KUKA KRL program: MyProgram_340().src

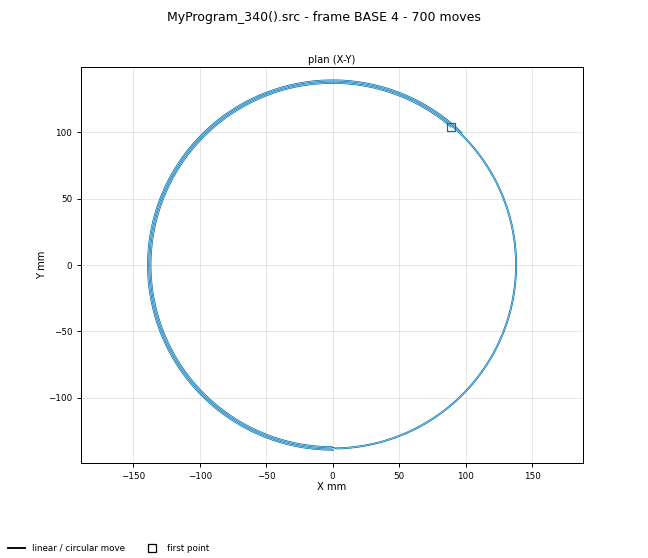
[picture p0: tool path of MyProgram_340().src in frame BASE 4, 700 of 700 moves have a stored position in this frame; points joined in program order, loops and branches not executed]
&ACCESS RVP
&REL 1
&PARAM TEMPLATE = C:\KRC\Roboter\Template\vorgabe
&PARAM EDITMASK = *
DEF MyProgram_340()
; ---- Setting reference (Base) ----
$BASE = BASE_DATA[4]

; --------------------------
; ---- Setting tool (TCP) ----
$TOOL = TOOL_DATA[3]
; --------------------------

$VEL.CP = VEL_APROX_PRINT
Startdeposition()
$VEL.CP = VEL_PRINT
LIN {X 89.0125,Y 103.7301,Z 191,A 47.9774,B 1.0012,C -0.0325,E1 1.1114,E2 406.47} C_DIS
LIN {X 85.5408,Y 106.6114,Z 191,A 49.6808,B 1.0011,C -0.0355,E1 1.1078,E2 404.7882} C_DIS
LIN {X 82.0051,Y 109.3546,Z 191,A 51.4263,B 1.001,C -0.0386,E1 1.1039,E2 403.0577} C_DIS
LIN {X 78.2991,Y 112.0376,Z 191,A 53.1641,B 1.0009,C -0.0415,E1 1.1,E2 401.3407} C_DIS
LIN {X 75.2781,Y 114.0891,Z 191,A 54.7295,B 1.0007,C -0.0444,E1 1.0963,E2 399.7713} C_DIS
LIN {X 72.4875,Y 115.8826,Z 191,A 55.8544,B 1.0007,C -0.0459,E1 1.0937,E2 398.6768} C_DIS
LIN {X 65.446,Y 119.9997,Z 191,A 58.9609,B 1.0005,C -0.0504,E1 1.0862,E2 395.6062} C_DIS
LIN {X 61.9887,Y 121.8193,Z 191,A 60.3832,B 1.0004,C -0.0523,E1 1.0827,E2 394.2083} C_DIS
LIN {X 59.3843,Y 123.111,Z 191,A 61.5861,B 1.0003,C -0.0541,E1 1.0796,E2 393.0073} C_DIS
LIN {X 56.2907,Y 124.556,Z 191,A 63.2488,B 1.0001,C -0.0571,E1 1.0753,E2 391.3188} C_DIS
LIN {X 52.6993,Y 126.1164,Z 191,A 64.3426,B 1.0001,C -0.0575,E1 1.0726,E2 390.2866} C_DIS
LIN {X 45.3684,Y 128.9368,Z 191,A 67.5319,B 0.9998,C -0.0616,E1 1.0643,E2 387.1097} C_DIS
LIN {X 41.7128,Y 130.1639,Z 191,A 68.9945,B 0.9998,C -0.0631,E1 1.0604,E2 385.6644} C_DIS
LIN {X 38.4614,Y 131.1614,Z 191,A 70.3424,B 0.9996,C -0.0645,E1 1.0567,E2 384.3254} C_DIS
LIN {X 34.8075,Y 132.1788,Z 191,A 71.8908,B 0.9996,C -0.0662,E1 1.0525,E2 382.7821} C_DIS
LIN {X 30.73,Y 133.1855,Z 191,A 73.5485,B 0.9994,C -0.0677,E1 1.048,E2 381.1362} C_DIS
LIN {X 27.316,Y 133.9271,Z 191,A 74.9001,B 0.9994,C -0.0688,E1 1.0443,E2 379.7974} C_DIS
LIN {X 24.0044,Y 134.5601,Z 191,A 76.1307,B 0.9994,C -0.0696,E1 1.041,E2 378.5872} C_DIS
LIN {X 21.0632,Y 135.0519,Z 191,A 77.6214,B 0.9992,C -0.0713,E1 1.0367,E2 377.0704} C_DIS
LIN {X 16.2963,Y 135.7096,Z 191,A 79.36,B 0.9992,C -0.0721,E1 1.0319,E2 375.3631} C_DIS
LIN {X 10.7417,Y 136.2638,Z 191,A 81.601,B 0.999,C -0.0735,E1 1.0257,E2 373.1338} C_DIS
LIN {X 3.1544,Y 136.6498,Z 191,A 84.6519,B 0.999,C -0.0749,E1 1.0171,E2 370.0986} C_DIS
LIN {X -4.6378,Y 136.6077,Z 191,A 88.9987,B 0.9986,C -0.0787,E1 1.0045,E2 365.6345} C_DIS
LIN {X -12.0307,Y 136.1551,Z 191,A 90.9637,B 0.9988,C -0.0769,E1 0.9993,E2 363.7961} C_DIS
LIN {X -15.8148,Y 135.7671,Z 191,A 92.6887,B 0.9988,C -0.0774,E1 0.9944,E2 362.0576} C_DIS
LIN {X -23.2946,Y 134.6872,Z 191,A 95.8708,B 0.9988,C -0.0774,E1 0.9855,E2 358.8755} C_DIS
LIN {X -27.1934,Y 133.9521,Z 191,A 97.4358,B 0.9988,C -0.0771,E1 0.9812,E2 357.3218} C_DIS
LIN {X -30.4676,Y 133.2454,Z 191,A 98.8461,B 0.9988,C -0.0769,E1 0.9773,E2 355.9115} C_DIS
LIN {X -34.0913,Y 132.3655,Z 191,A 100.4982,B 0.9988,C -0.0766,E1 0.9727,E2 354.2506} C_DIS
LIN {X -38.1454,Y 131.254,Z 191,A 102.2716,B 0.9988,C -0.0761,E1 0.9679,E2 352.4768} C_DIS
LIN {X -41.8854,Y 130.1088,Z 191,A 103.6911,B 0.9989,C -0.0751,E1 0.9642,E2 351.0819} C_DIS
LIN {X -46.7376,Y 128.4459,Z 191,A 106.4411,B 0.9989,C -0.0748,E1 0.9567,E2 348.2678} C_DIS
LIN {X -50.0052,Y 127.2098,Z 191,A 107.7565,B 0.999,C -0.0737,E1 0.9532,E2 346.9696} C_DIS
LIN {X -54.4673,Y 125.3632,Z 191,A 110.0747,B 0.999,C -0.0726,E1 0.9471,E2 344.6202} C_DIS
LIN {X -57.7457,Y 123.8877,Z 191,A 111.3528,B 0.9992,C -0.0712,E1 0.9439,E2 343.368} C_DIS
LIN {X -61.7186,Y 121.9568,Z 191,A 113.2508,B 0.9993,C -0.0696,E1 0.9391,E2 341.4659} C_DIS
LIN {X -65.1433,Y 120.1648,Z 191,A 115.3058,B 0.9993,C -0.0685,E1 0.9339,E2 339.3641} C_DIS
LIN {X -68.2953,Y 118.4015,Z 191,A 116.6428,B 0.9995,C -0.0668,E1 0.9306,E2 338.0475} C_DIS
LIN {X -71.0356,Y 116.7783,Z 191,A 118.4141,B 0.9995,C -0.0656,E1 0.9263,E2 336.2288} C_DIS
LIN {X -74.4665,Y 114.6204,Z 191,A 119.7536,B 0.9997,C -0.0634,E1 0.9232,E2 334.93} C_DIS
LIN {X -77.8426,Y 112.3553,Z 191,A 121.5206,B 0.9998,C -0.0613,E1 0.919,E2 333.1571} C_DIS
LIN {X -80.4484,Y 110.5045,Z 191,A 123.3051,B 0.9999,C -0.0597,E1 0.9149,E2 331.3241} C_DIS
LIN {X -86.3086,Y 105.9905,Z 191,A 126.4807,B 1.0002,C -0.0553,E1 0.9078,E2 328.1421} C_DIS
LIN {X -88.7872,Y 103.9233,Z 191,A 128.3952,B 1.0002,C -0.0534,E1 0.9036,E2 326.1654} C_DIS
LIN {X -92.1512,Y 100.9523,Z 191,A 129.7061,B 1.0005,C -0.0503,E1 0.901,E2 324.9197} C_DIS
LIN {X -97.6119,Y 95.6818,Z 191,A 133.23,B 1.0007,C -0.0449,E1 0.8938,E2 321.3597} C_DIS
LIN {X -100.937,Y 92.1667,Z 191,A 135.8857,B 1.0009,C -0.0412,E1 0.8886,E2 318.6342} C_DIS
LIN {X -106.4904,Y 85.6908,Z 191,A 139.6872,B 1.0011,C -0.0342,E1 0.8816,E2 314.8093} C_DIS
LIN {X -108.7863,Y 82.7573,Z 191,A 141.3018,B 1.0012,C -0.0311,E1 0.8789,E2 313.1896} C_DIS
LIN {X -111.015,Y 79.7425,Z 191,A 143.212,B 1.0013,C -0.0277,E1 0.8756,E2 311.2413} C_DIS
LIN {X -113.3974,Y 76.3169,Z 191,A 145.1171,B 1.0014,C -0.0239,E1 0.8726,E2 309.3194} C_DIS
LIN {X -115.7378,Y 72.7183,Z 191,A 147.066,B 1.0015,C -0.0198,E1 0.8696,E2 307.3543} C_DIS
LIN {X -118.0316,Y 68.9321,Z 191,A 149.3442,B 1.0016,C -0.0154,E1 0.8663,E2 305.0279} C_DIS
LIN {X -119.6578,Y 66.0693,Z 191,A 151.1723,B 1.0016,C -0.0119,E1 0.8637,E2 303.1479} C_DIS
LIN {X -121.3639,Y 62.8801,Z 191,A 152.6426,B 1.0016,C -0.0084,E1 0.8618,E2 301.684} C_DIS
LIN {X -122.9907,Y 59.6361,Z 191,A 154.354,B 1.0017,C -0.0046,E1 0.8597,E2 299.951} C_DIS
LIN {X -124.7758,Y 55.7992,Z 191,A 156.2284,B 1.0017,C -0.0001,E1 0.8575,E2 298.0657} C_DIS
LIN {X -126.2515,Y 52.3759,Z 191,A 158.1097,B 1.0017,C 0.004,E1 0.8554,E2 296.1474} C_DIS
LIN {X -127.8965,Y 48.2198,Z 191,A 160.229,B 1.0017,C 0.0089,E1 0.8532,E2 293.9998} C_DIS
LIN {X -129.0749,Y 44.9701,Z 191,A 161.9157,B 1.0017,C 0.0129,E1 0.8516,E2 292.2853} C_DIS
LIN {X -130.2137,Y 41.5569,Z 191,A 163.6416,B 1.0016,C 0.017,E1 0.8501,E2 290.534} C_DIS
LIN {X -131.1238,Y 38.5898,Z 191,A 165.1276,B 1.0016,C 0.0206,E1 0.8489,E2 289.0263} C_DIS
LIN {X -131.9252,Y 35.7585,Z 191,A 166.5518,B 1.0014,C 0.024,E1 0.8478,E2 287.5796} C_DIS
LIN {X -132.8248,Y 32.2526,Z 191,A 168.7786,B 1.0014,C 0.0287,E1 0.8463,E2 285.2663} C_DIS
LIN {X -133.6596,Y 28.5972,Z 191,A 170.156,B 1.0012,C 0.0328,E1 0.8455,E2 283.9139} C_DIS
LIN {X -134.4207,Y 24.7837,Z 191,A 172.2093,B 1.001,C 0.0376,E1 0.8444,E2 281.8092} C_DIS
LIN {X -135.0064,Y 21.3572,Z 191,A 173.7372,B 1.0009,C 0.0417,E1 0.8437,E2 280.2733} C_DIS
LIN {X -135.4771,Y 18.1315,Z 191,A 175.4147,B 1.0007,C 0.0458,E1 0.843,E2 278.5578} C_DIS
LIN {X -135.9257,Y 14.3847,Z 191,A 177.2703,B 1.0005,C 0.0504,E1 0.8424,E2 276.6687} C_DIS
LIN {X -136.3047,Y 10.1866,Z 191,A 179.2613,B 1.0002,C 0.0555,E1 0.842,E2 274.6504} C_DIS
LIN {X -136.5247,Y 6.6162,Z 191,A -178.9262,B 0.9999,C 0.06,E1 0.8417,E2 272.7991} C_DIS
LIN {X -136.6594,Y 2.6599,Z 191,A -177.0143,B 0.9996,C 0.0649,E1 0.8416,E2 270.856} C_DIS
LIN {X -136.6818,Y -1.0196,Z 191,A -175.0654,B 0.9993,C 0.0695,E1 0.8416,E2 268.8557} C_DIS
LIN {X -136.5818,Y -5.3018,Z 191,A -173.1233,B 0.9989,C 0.0747,E1 0.8417,E2 266.8957} C_DIS
LIN {X -136.3676,Y -9.3245,Z 191,A -171.0934,B 0.9985,C 0.0797,E1 0.8421,E2 264.8227} C_DIS
LIN {X -136.054,Y -13.1141,Z 191,A -169.2581,B 0.9982,C 0.0843,E1 0.8426,E2 262.9567} C_DIS
LIN {X -135.5716,Y -17.4107,Z 191,A -167.1462,B 0.9977,C 0.0896,E1 0.8433,E2 260.8066} C_DIS
LIN {X -135.0756,Y -20.9104,Z 191,A -165.3797,B 0.9973,C 0.0939,E1 0.844,E2 259.0034} C_DIS
LIN {X -134.3255,Y -25.287,Z 191,A -163.2215,B 0.9968,C 0.0992,E1 0.8451,E2 256.807} C_DIS
LIN {X -133.6562,Y -28.6131,Z 191,A -161.7639,B 0.9964,C 0.103,E1 0.8459,E2 255.3453} C_DIS
LIN {X -132.915,Y -31.8785,Z 191,A -160.1593,B 0.996,C 0.107,E1 0.847,E2 253.7147} C_DIS
LIN {X -132.2033,Y -34.7156,Z 191,A -158.4885,B 0.9956,C 0.1105,E1 0.8482,E2 251.9852} C_DIS
LIN {X -131.2438,Y -38.18,Z 191,A -156.9119,B 0.9952,C 0.1145,E1 0.8494,E2 250.4} C_DIS
LIN {X -130.259,Y -41.4151,Z 191,A -155.3551,B 0.9947,C 0.1183,E1 0.8507,E2 248.825} C_DIS
LIN {X -129.3087,Y -44.2956,Z 191,A -153.8993,B 0.9943,C 0.1217,E1 0.852,E2 247.345} C_DIS
LIN {X -127.3684,Y -49.597,Z 191,A -151.0547,B 0.9935,C 0.128,E1 0.8548,E2 244.4368} C_DIS
LIN {X -126.0875,Y -52.7686,Z 191,A -149.3641,B 0.993,C 0.1317,E1 0.8567,E2 242.7118} C_DIS
LIN {X -124.7202,Y -55.9236,Z 191,A -147.7644,B 0.9925,C 0.1353,E1 0.8585,E2 241.0911} C_DIS
LIN {X -123.4648,Y -58.6438,Z 191,A -146.2796,B 0.9921,C 0.1384,E1 0.8603,E2 239.5754} C_DIS
LIN {X -121.9116,Y -61.8075,Z 191,A -144.679,B 0.9916,C 0.142,E1 0.8623,E2 237.9583} C_DIS
LIN {X -120.1841,Y -65.1061,Z 191,A -142.4979,B 0.9911,C 0.1458,E1 0.8653,E2 235.6923} C_DIS
LIN {X -118.5495,Y -68.0385,Z 191,A -141.1245,B 0.9906,C 0.1489,E1 0.8672,E2 234.3241} C_DIS
LIN {X -116.0458,Y -72.2251,Z 191,A -138.8268,B 0.9899,C 0.1535,E1 0.8706,E2 231.9918} C_DIS
LIN {X -113.6068,Y -76.0041,Z 191,A -136.7006,B 0.9892,C 0.1576,E1 0.874,E2 229.8325} C_DIS
LIN {X -111.2543,Y -79.4078,Z 191,A -134.7546,B 0.9887,C 0.1612,E1 0.8772,E2 227.8574} C_DIS
LIN {X -108.5406,Y -83.0786,Z 191,A -132.6287,B 0.988,C 0.1651,E1 0.8808,E2 225.7021} C_DIS
LIN {X -105.6615,Y -86.7112,Z 191,A -130.4933,B 0.9874,C 0.1688,E1 0.8846,E2 223.54} C_DIS
LIN {X -102.7803,Y -90.1077,Z 191,A -128.4742,B 0.9868,C 0.1723,E1 0.8883,E2 221.4997} C_DIS
LIN {X -99.9949,Y -93.1886,Z 191,A -126.4868,B 0.9863,C 0.1753,E1 0.8922,E2 219.4776} C_DIS
LIN {X -96.802,Y -96.5015,Z 191,A -124.4491,B 0.9857,C 0.1786,E1 0.8962,E2 217.4246} C_DIS
LIN {X -91.9919,Y -101.0971,Z 191,A -121.3065,B 0.9849,C 0.1829,E1 0.9028,E2 214.232} C_DIS
LIN {X -88.5887,Y -104.092,Z 191,A -119.2485,B 0.9844,C 0.1857,E1 0.9072,E2 212.1516} C_DIS
LIN {X -85.0432,Y -107.0083,Z 191,A -117.1981,B 0.9839,C 0.1883,E1 0.9117,E2 210.0831} C_DIS
LIN {X -81.4237,Y -109.7877,Z 191,A -115.1197,B 0.9834,C 0.1907,E1 0.9165,E2 207.981} C_DIS
LIN {X -78.6696,Y -111.7775,Z 191,A -112.9292,B 0.9832,C 0.1917,E1 0.9218,E2 205.6802} C_DIS
LIN {X -74.0073,Y -114.918,Z 191,A -110.2765,B 0.9828,C 0.194,E1 0.9282,E2 202.9843} C_DIS
LIN {X -68.59,Y -118.2308,Z 191,A -108.2796,B 0.982,C 0.1977,E1 0.9328,E2 201.0832} C_DIS
LIN {X -64.6067,Y -120.4537,Z 191,A -106.1921,B 0.9817,C 0.1992,E1 0.9381,E2 198.9701} C_DIS
LIN {X -60.9145,Y -122.361,Z 191,A -104.507,B 0.9814,C 0.2008,E1 0.9423,E2 197.2928} C_DIS
LIN {X -55.0681,Y -125.1029,Z 191,A -101.7411,B 0.981,C 0.2028,E1 0.9494,E2 194.5179} C_DIS
LIN {X -48.4203,Y -127.8214,Z 191,A -98.6538,B 0.9806,C 0.2045,E1 0.9576,E2 191.4188} C_DIS
LIN {X -45.2797,Y -128.9675,Z 191,A -97.2652,B 0.9805,C 0.2052,E1 0.9612,E2 190.0317} C_DIS
LIN {X -41.8249,Y -130.1281,Z 191,A -95.648,B 0.9804,C 0.2057,E1 0.9656,E2 188.401} C_DIS
LIN {X -38.4661,Y -131.1601,Z 191,A -94.1345,B 0.9803,C 0.2062,E1 0.9697,E2 186.8811} C_DIS
LIN {X -35.798,Y -131.9146,Z 191,A -92.8618,B 0.9803,C 0.2062,E1 0.9732,E2 185.5921} C_DIS
LIN {X -32.0236,Y -132.88,Z 191,A -91.2701,B 0.9802,C 0.2067,E1 0.9776,E2 184.0058} C_DIS
LIN {X -28.5972,Y -133.6596,Z 191,A -89.7763,B 0.9802,C 0.2069,E1 0.9817,E2 182.5084} C_DIS
LIN {X -25.9354,Y -134.2016,Z 191,A -88.4583,B 0.9802,C 0.2066,E1 0.9855,E2 181.1639} C_DIS
LIN {X -20.2685,Y -135.175,Z 191,A -86.2694,B 0.9801,C 0.2071,E1 0.9915,E2 179.0062} C_DIS
LIN {X -15.9902,Y -135.7462,Z 191,A -84.4316,B 0.9801,C 0.2069,E1 0.9967,E2 177.1633} C_DIS
LIN {X -13.182,Y -136.0475,Z 191,A -82.9996,B 0.9803,C 0.206,E1 1.0008,E2 175.6947} C_DIS
LIN {X -7.968,Y -136.4529,Z 191,A -80.9818,B 0.9803,C 0.2059,E1 1.0064,E2 173.7012} C_DIS
LIN {X -0.5095,Y -136.684,Z 191,A -78.0357,B 0.9805,C 0.2052,E1 1.0147,E2 170.78} C_DIS
LIN {X -0.5095,Y -136.684,Z 191,A -78.0358,B 0.9805,C 0.2052,E1 1.0147,E2 170.7801} C_DIS
Enddeposition()
LIN {X 0.9755,Y -137.5796,Z 191,A -77.8874,B 0.9714,C 0.2064,E1 1.0061,E2 170.7271} C_DIS
Startdeposition()
$VEL.CP = VEL_PRINT
LIN {X -2.3504,Y -137.5636,Z 191,A -79.4321,B 0.9712,C 0.2074,E1 1.0017,E2 172.2957} C_DIS
LIN {X -6.1614,Y -137.4476,Z 191,A -80.9814,B 0.9712,C 0.2079,E1 0.9973,E2 173.8404} C_DIS
LIN {X -10.1773,Y -137.2067,Z 191,A -82.5541,B 0.9711,C 0.208,E1 0.9929,E2 175.3989} C_DIS
LIN {X -14.2933,Y -136.8397,Z 191,A -84.3553,B 0.971,C 0.2086,E1 0.9878,E2 177.2126} C_DIS
LIN {X -20.3097,Y -136.0782,Z 191,A -86.6928,B 0.971,C 0.2083,E1 0.9813,E2 179.524} C_DIS
LIN {X -26.9326,Y -134.9225,Z 191,A -89.4105,B 0.971,C 0.208,E1 0.9738,E2 182.231} C_DIS
LIN {X -30.869,Y -134.0758,Z 191,A -91.1981,B 0.971,C 0.208,E1 0.9688,E2 184.0353} C_DIS
LIN {X -34.03,Y -133.3085,Z 191,A -92.6122,B 0.9711,C 0.2079,E1 0.9649,E2 185.4586} C_DIS
LIN {X -37.2832,Y -132.4355,Z 191,A -94.0679,B 0.9711,C 0.2076,E1 0.9609,E2 186.9225} C_DIS
LIN {X -40.6978,Y -131.4269,Z 191,A -95.5338,B 0.9713,C 0.207,E1 0.9569,E2 188.3864} C_DIS
LIN {X -43.6182,Y -130.486,Z 191,A -96.8165,B 0.9714,C 0.2064,E1 0.9535,E2 189.6703} C_DIS
LIN {X -46.7356,Y -129.4021,Z 191,A -98.3193,B 0.9715,C 0.206,E1 0.9494,E2 191.1921} C_DIS
LIN {X -50.5842,Y -127.9491,Z 191,A -100.2988,B 0.9716,C 0.2055,E1 0.9441,E2 193.2105} C_DIS
LIN {X -54.8307,Y -126.1854,Z 191,A -101.9447,B 0.972,C 0.2038,E1 0.9399,E2 194.818} C_DIS
LIN {X -57.6498,Y -124.9224,Z 191,A -103.437,B 0.9721,C 0.2031,E1 0.936,E2 196.3404} C_DIS
LIN {X -61.24,Y -123.2028,Z 191,A -105.0696,B 0.9724,C 0.2018,E1 0.9319,E2 197.9697} C_DIS
LIN {X -64.6588,Y -121.4452,Z 191,A -106.8458,B 0.9727,C 0.2006,E1 0.9274,E2 199.7715} C_DIS
LIN {X -68.4652,Y -119.3411,Z 191,A -108.7461,B 0.973,C 0.1989,E1 0.9226,E2 201.6849} C_DIS
LIN {X -73.0298,Y -116.6039,Z 191,A -111.0777,B 0.9734,C 0.1967,E1 0.917,E2 204.0335} C_DIS
LIN {X -76.7762,Y -114.172,Z 191,A -113.3045,B 0.9738,C 0.1949,E1 0.9116,E2 206.313} C_DIS
LIN {X -79.5332,Y -112.2684,Z 191,A -114.5548,B 0.9742,C 0.193,E1 0.9088,E2 207.5427} C_DIS
LIN {X -82.9847,Y -109.7415,Z 191,A -116.466,B 0.9746,C 0.1908,E1 0.9044,E2 209.4725} C_DIS
LIN {X -86.4102,Y -107.0651,Z 191,A -118.4124,B 0.9751,C 0.1883,E1 0.9001,E2 211.4383} C_DIS
LIN {X -89.5447,Y -104.4581,Z 191,A -120.3137,B 0.9755,C 0.186,E1 0.8959,E2 213.3686} C_DIS
LIN {X -93.0211,Y -101.3742,Z 191,A -122.5042,B 0.9761,C 0.1831,E1 0.8913,E2 215.5953} C_DIS
LIN {X -96.7246,Y -97.8475,Z 191,A -124.6857,B 0.9767,C 0.1796,E1 0.8868,E2 217.7841} C_DIS
LIN {X -99.6065,Y -94.9117,Z 191,A -126.588,B 0.9773,C 0.1767,E1 0.8831,E2 219.7129} C_DIS
LIN {X -102.6845,Y -91.573,Z 191,A -128.6464,B 0.9779,C 0.1734,E1 0.8791,E2 221.7946} C_DIS
LIN {X -105.6134,Y -88.1791,Z 191,A -130.7495,B 0.9785,C 0.1699,E1 0.8752,E2 223.9307} C_DIS
LIN {X -108.4646,Y -84.6479,Z 191,A -132.8938,B 0.9791,C 0.1662,E1 0.8714,E2 226.1104} C_DIS
LIN {X -111.2531,Y -80.9472,Z 191,A -135.0363,B 0.9798,C 0.1623,E1 0.8678,E2 228.2822} C_DIS
LIN {X -113.8906,Y -77.1919,Z 191,A -137.175,B 0.9804,C 0.1583,E1 0.8643,E2 230.4522} C_DIS
LIN {X -116.3526,Y -73.4284,Z 191,A -139.3153,B 0.9811,C 0.1542,E1 0.861,E2 232.629} C_DIS
LIN {X -119.0033,Y -69.0499,Z 191,A -142.5443,B 0.9818,C 0.1492,E1 0.8563,E2 236.0081} C_DIS
LIN {X -121.9972,Y -63.6076,Z 191,A -144.5104,B 0.9827,C 0.1433,E1 0.8538,E2 237.8887} C_DIS
LIN {X -123.5368,Y -60.5629,Z 191,A -146.1854,B 0.9832,C 0.1399,E1 0.8516,E2 239.598} C_DIS
LIN {X -125.253,Y -56.9339,Z 191,A -148.2535,B 0.9838,C 0.1356,E1 0.8491,E2 241.7196} C_DIS
LIN {X -127.0422,Y -52.8152,Z 191,A -150.2585,B 0.9844,C 0.131,E1 0.8469,E2 243.7423} C_DIS
LIN {X -128.8535,Y -48.2274,Z 191,A -152.6351,B 0.9851,C 0.1256,E1 0.8445,E2 246.1617} C_DIS
LIN {X -130.1279,Y -44.6768,Z 191,A -154.3839,B 0.9857,C 0.1215,E1 0.8428,E2 247.9338} C_DIS
LIN {X -131.161,Y -41.5458,Z 191,A -155.925,B 0.9861,C 0.1178,E1 0.8415,E2 249.4969} C_DIS
LIN {X -132.1072,Y -38.4304,Z 191,A -157.5422,B 0.9865,C 0.1141,E1 0.8402,E2 251.1486} C_DIS
LIN {X -133.1124,Y -34.795,Z 191,A -159.3155,B 0.987,C 0.1098,E1 0.8389,E2 252.9482} C_DIS
LIN {X -133.7924,Y -32.0747,Z 191,A -160.6918,B 0.9874,C 0.1065,E1 0.8379,E2 254.3516} C_DIS
LIN {X -134.4829,Y -29.0433,Z 191,A -162.235,B 0.9878,C 0.1028,E1 0.837,E2 255.9272} C_DIS
LIN {X -135.2705,Y -25.1312,Z 191,A -164.3349,B 0.9883,C 0.098,E1 0.8358,E2 258.084} C_DIS
LIN {X -135.9783,Y -20.9551,Z 191,A -166.1966,B 0.9887,C 0.0931,E1 0.835,E2 259.9576} C_DIS
LIN {X -136.4504,Y -17.6228,Z 191,A -167.9204,B 0.9891,C 0.0889,E1 0.8343,E2 261.7228} C_DIS
LIN {X -136.9391,Y -13.301,Z 191,A -170.0176,B 0.9896,C 0.0837,E1 0.8337,E2 263.8562} C_DIS
LIN {X -137.2547,Y -9.5192,Z 191,A -171.9652,B 0.99,C 0.079,E1 0.8333,E2 265.8505} C_DIS
LIN {X -137.4766,Y -5.4259,Z 191,A -173.8399,B 0.9904,C 0.074,E1 0.833,E2 267.7458} C_DIS
LIN {X -137.5778,Y -1.4513,Z 191,A -175.8623,B 0.9907,C 0.0691,E1 0.833,E2 269.8142} C_DIS
LIN {X -137.5571,Y 2.7372,Z 191,A -177.8981,B 0.9911,C 0.0639,E1 0.833,E2 271.8861} C_DIS
LIN {X -137.416,Y 6.7903,Z 191,A -179.8134,B 0.9914,C 0.059,E1 0.8332,E2 273.8291} C_DIS
LIN {X -137.1733,Y 10.6343,Z 191,A 178.1911,B 0.9916,C 0.0542,E1 0.8336,E2 275.873} C_DIS
LIN {X -136.7905,Y 14.7502,Z 191,A 176.3408,B 0.9919,C 0.0493,E1 0.8341,E2 277.7383} C_DIS
LIN {X -136.3259,Y 18.5724,Z 191,A 174.2864,B 0.9921,C 0.0444,E1 0.8349,E2 279.848} C_DIS
LIN {X -135.7059,Y 22.6516,Z 191,A 172.4219,B 0.9923,C 0.0395,E1 0.8357,E2 281.7295} C_DIS
LIN {X -135.0578,Y 26.244,Z 191,A 170.6382,B 0.9925,C 0.0351,E1 0.8367,E2 283.5448} C_DIS
LIN {X -134.107,Y 30.7327,Z 191,A 168.39,B 0.9927,C 0.0297,E1 0.838,E2 285.8333} C_DIS
LIN {X -133.0599,Y 34.9919,Z 191,A 166.3658,B 0.9928,C 0.0246,E1 0.8394,E2 287.8805} C_DIS
LIN {X -132.1069,Y 38.4315,Z 191,A 164.4992,B 0.9929,C 0.0203,E1 0.8409,E2 289.7922} C_DIS
LIN {X -130.9132,Y 42.3214,Z 191,A 162.6742,B 0.9929,C 0.0157,E1 0.8424,E2 291.632} C_DIS
LIN {X -129.86,Y 45.4498,Z 191,A 161.0565,B 0.993,C 0.012,E1 0.8439,E2 293.278} C_DIS
LIN {X -128.7512,Y 48.5005,Z 191,A 159.4542,B 0.993,C 0.0083,E1 0.8455,E2 294.9094} C_DIS
LIN {X -127.3455,Y 52.0838,Z 191,A 157.6483,B 0.9931,C 0.0041,E1 0.8474,E2 296.7386} C_DIS
LIN {X -125.8846,Y 55.5219,Z 191,A 155.6562,B 0.9931,C -0.0001,E1 0.8497,E2 298.7813} C_DIS
LIN {X -123.9004,Y 59.8173,Z 191,A 153.6151,B 0.9931,C -0.0049,E1 0.8521,E2 300.8295} C_DIS
LIN {X -122.4671,Y 62.6977,Z 191,A 152.0069,B 0.9931,C -0.0083,E1 0.8542,E2 302.4682} C_DIS
LIN {X -120.1746,Y 66.9917,Z 191,A 149.6109,B 0.9931,C -0.0133,E1 0.8575,E2 304.906} C_DIS
LIN {X -117.1207,Y 72.1975,Z 191,A 146.7692,B 0.9929,C -0.0191,E1 0.8616,E2 307.7841} C_DIS
LIN {X -114.6585,Y 76.0476,Z 191,A 144.6065,B 0.9929,C -0.0234,E1 0.865,E2 309.9754} C_DIS
LIN {X -112.1096,Y 79.7571,Z 191,A 142.5051,B 0.9927,C -0.0275,E1 0.8684,E2 312.1015} C_DIS
LIN {X -108.8533,Y 84.1466,Z 191,A 140.1427,B 0.9926,C -0.0322,E1 0.8724,E2 314.4724} C_DIS
LIN {X -105.323,Y 88.5252,Z 191,A 137.2526,B 0.9924,C -0.0369,E1 0.8776,E2 317.423} C_DIS
LIN {X -102.4692,Y 91.8135,Z 191,A 134.6875,B 0.9923,C -0.0404,E1 0.8826,E2 320.0708} C_DIS
LIN {X -98.7949,Y 95.7561,Z 191,A 133.367,B 0.9921,C -0.0444,E1 0.885,E2 321.2868} C_DIS
LIN {X -95.3607,Y 99.1774,Z 191,A 130.6309,B 0.992,C -0.0478,E1 0.8906,E2 324.102} C_DIS
LIN {X -91.3994,Y 102.839,Z 191,A 127.6625,B 0.9918,C -0.0513,E1 0.897,E2 327.1485} C_DIS
LIN {X -87.7377,Y 105.9799,Z 191,A 126.1159,B 0.9916,C -0.0544,E1 0.9002,E2 328.6432} C_DIS
LIN {X -82.2759,Y 110.274,Z 191,A 122.4127,B 0.9914,C -0.0582,E1 0.9087,E2 332.4332} C_DIS
LIN {X -78.5502,Y 112.958,Z 191,A 120.9733,B 0.9913,C -0.0608,E1 0.9119,E2 333.82} C_DIS
LIN {X -75.2948,Y 115.1544,Z 191,A 119.0116,B 0.9911,C -0.0626,E1 0.9166,E2 335.8164} C_DIS
LIN {X -71.5352,Y 117.5267,Z 191,A 117.0965,B 0.9911,C -0.0647,E1 0.9212,E2 337.7373} C_DIS
LIN {X -67.6499,Y 119.8049,Z 191,A 115.1076,B 0.9909,C -0.0665,E1 0.9261,E2 339.7375} C_DIS
LIN {X -63.7058,Y 121.9456,Z 191,A 113.2532,B 0.9908,C -0.0683,E1 0.9307,E2 341.5891} C_DIS
LIN {X -60.3355,Y 123.649,Z 191,A 111.5289,B 0.9907,C -0.0695,E1 0.9351,E2 343.3291} C_DIS
LIN {X -56.6215,Y 125.3928,Z 191,A 109.2716,B 0.9907,C -0.0702,E1 0.9411,E2 345.6442} C_DIS
LIN {X -52.2336,Y 127.2849,Z 191,A 107.7938,B 0.9905,C -0.0721,E1 0.9448,E2 347.0662} C_DIS
LIN {X -48.6101,Y 128.7102,Z 191,A 105.2683,B 0.9905,C -0.072,E1 0.9517,E2 349.6873} C_DIS
LIN {X -42.8275,Y 130.7493,Z 191,A 103.5296,B 0.9903,C -0.0743,E1 0.9561,E2 351.338} C_DIS
LIN {X -39.9991,Y 131.6407,Z 191,A 102.1985,B 0.9903,C -0.0746,E1 0.9597,E2 352.6787} C_DIS
LIN {X -36.7199,Y 132.593,Z 191,A 100.8049,B 0.9903,C -0.0752,E1 0.9635,E2 354.0685} C_DIS
LIN {X -33.2062,Y 133.5176,Z 191,A 99.2577,B 0.9903,C -0.0755,E1 0.9678,E2 355.6187} C_DIS
LIN {X -30.1359,Y 134.2433,Z 191,A 97.9714,B 0.9903,C -0.0758,E1 0.9713,E2 356.9015} C_DIS
LIN {X -27.1204,Y 134.8843,Z 191,A 96.6055,B 0.9903,C -0.0758,E1 0.9751,E2 358.2755} C_DIS
LIN {X -22.8887,Y 135.6664,Z 191,A 94.6325,B 0.9903,C -0.0756,E1 0.9807,E2 360.2671} C_DIS
LIN {X -16.2805,Y 136.6168,Z 191,A 92.0873,B 0.9903,C -0.0758,E1 0.9877,E2 362.7859} C_DIS
LIN {X -12.9872,Y 136.9693,Z 191,A 90.7086,B 0.9903,C -0.0756,E1 0.9916,E2 364.1639} C_DIS
LIN {X -9.1202,Y 137.2825,Z 191,A 88.5737,B 0.9903,C -0.0741,E1 0.9978,E2 366.3537} C_DIS
LIN {X -4.5471,Y 137.5104,Z 191,A 87.2726,B 0.9903,C -0.0748,E1 1.0013,E2 367.5893} C_DIS
LIN {X 2.4832,Y 137.5614,Z 191,A 84.4448,B 0.9903,C -0.0737,E1 1.0093,E2 370.4052} C_DIS
LIN {X 5.7855,Y 137.4626,Z 191,A 83.0466,B 0.9904,C -0.073,E1 1.0132,E2 371.8053} C_DIS
LIN {X 8.6467,Y 137.3117,Z 191,A 81.8644,B 0.9904,C -0.0723,E1 1.0165,E2 372.9859} C_DIS
LIN {X 12.6768,Y 136.9991,Z 191,A 80.0333,B 0.9906,C -0.0708,E1 1.0217,E2 374.8324} C_DIS
LIN {X 17.0816,Y 136.5213,Z 191,A 78.4841,B 0.9906,C -0.0702,E1 1.026,E2 376.3492} C_DIS
LIN {X 23.4637,Y 135.5701,Z 191,A 75.9145,B 0.9908,C -0.0682,E1 1.0331,E2 378.9053} C_DIS
LIN {X 27.2464,Y 134.8586,Z 191,A 74.3537,B 0.9908,C -0.0668,E1 1.0375,E2 380.461} C_DIS
LIN {X 30.6029,Y 134.1366,Z 191,A 72.9821,B 0.9909,C -0.0656,E1 1.0412,E2 381.8258} C_DIS
LIN {X 34.149,Y 133.2783,Z 191,A 71.5276,B 0.991,C -0.0641,E1 1.0452,E2 383.2728} C_DIS
LIN {X 37.5501,Y 132.3609,Z 191,A 70.2116,B 0.9911,C -0.0629,E1 1.0487,E2 384.572} C_DIS
LIN {X 40.3296,Y 131.5396,Z 191,A 69.0293,B 0.9912,C -0.0616,E1 1.0519,E2 385.7513} C_DIS
LIN {X 43.6605,Y 130.472,Z 191,A 67.6613,B 0.9912,C -0.0601,E1 1.0555,E2 387.1093} C_DIS
LIN {X 47.3979,Y 129.163,Z 191,A 65.88,B 0.9915,C -0.0574,E1 1.0603,E2 388.9049} C_DIS
LIN {X 51.5423,Y 127.5638,Z 191,A 64.4,B 0.9915,C -0.0561,E1 1.0641,E2 390.3436} C_DIS
LIN {X 55.1122,Y 126.0637,Z 191,A 62.8498,B 0.9916,C -0.054,E1 1.0681,E2 391.8868} C_DIS
LIN {X 58.025,Y 124.7489,Z 191,A 61.6509,B 0.9917,C -0.0525,E1 1.0711,E2 393.0708} C_DIS
LIN {X 61.331,Y 123.1579,Z 191,A 60.2491,B 0.9918,C -0.0506,E1 1.0746,E2 394.4583} C_DIS
LIN {X 65.1031,Y 121.2074,Z 191,A 58.5274,B 0.992,C -0.0479,E1 1.0789,E2 396.1747} C_DIS
LIN {X 69.6354,Y 118.6616,Z 191,A 56.7498,B 0.992,C -0.0457,E1 1.0832,E2 397.9087} C_DIS
LIN {X 72.4509,Y 116.9641,Z 191,A 55.2563,B 0.9922,C -0.0428,E1 1.0868,E2 399.4161} C_DIS
LIN {X 76.2951,Y 114.4933,Z 191,A 53.5365,B 0.9923,C -0.0401,E1 1.0908,E2 401.1151} C_DIS
LIN {X 80.1583,Y 111.8227,Z 191,A 51.7644,B 0.9924,C -0.0371,E1 1.0948,E2 402.8663} C_DIS
LIN {X 83.872,Y 109.0655,Z 191,A 50.0063,B 0.9925,C -0.0341,E1 1.0987,E2 404.6054} C_DIS
LIN {X 87.2973,Y 106.3434,Z 191,A 48.3731,B 0.9926,C -0.0312,E1 1.1022,E2 406.2171} C_DIS
LIN {X 90.7316,Y 103.429,Z 191,A 46.6587,B 0.9927,C -0.0281,E1 1.1058,E2 407.9131} C_DIS
LIN {X 93.954,Y 100.5105,Z 191,A 45.0724,B 0.9927,C -0.0252,E1 1.1091,E2 409.4737} C_DIS
LIN {X 97.0603,Y 97.5139,Z 191,A 43.4133,B 0.9929,C -0.022,E1 1.1124,E2 411.1169} C_DIS
LIN {X 100.2727,Y 94.2078,Z 191,A 41.6823,B 0.9929,C -0.0186,E1 1.1157,E2 412.8262} C_DIS
LIN {X 103.2679,Y 90.9146,Z 191,A 40.02,B 0.9929,C -0.0152,E1 1.1188,E2 414.4664} C_DIS
LIN {X 106.2288,Y 87.4372,Z 191,A 38.3589,B 0.993,C -0.0119,E1 1.1217,E2 416.0996} C_DIS
LIN {X 108.9095,Y 84.074,Z 191,A 36.7417,B 0.993,C -0.0085,E1 1.1245,E2 417.6966} C_DIS
LIN {X 111.5028,Y 80.6027,Z 191,A 35.1119,B 0.9931,C -0.0051,E1 1.1271,E2 419.3062} C_DIS
LIN {X 114.1371,Y 76.8277,Z 191,A 33.349,B 0.9931,C -0.0011,E1 1.1299,E2 421.0512} C_DIS
LIN {X 116.5474,Y 73.1198,Z 191,A 31.7983,B 0.9931,C 0.002,E1 1.1322,E2 422.5676} C_DIS
LIN {X 118.8132,Y 69.3773,Z 191,A 30.1058,B 0.9931,C 0.006,E1 1.1346,E2 424.2451} C_DIS
LIN {X 121.0286,Y 65.436,Z 191,A 28.4668,B 0.9931,C 0.0096,E1 1.1368,E2 425.8554} C_DIS
LIN {X 122.9821,Y 61.6861,Z 191,A 26.9917,B 0.9931,C 0.0127,E1 1.1386,E2 427.2964} C_DIS
LIN {X 124.757,Y 58.0074,Z 191,A 25.3815,B 0.993,C 0.0166,E1 1.1405,E2 428.8961} C_DIS
LIN {X 126.6075,Y 53.8546,Z 191,A 23.8342,B 0.993,C 0.0199,E1 1.1422,E2 430.402} C_DIS
LIN {X 128.1012,Y 50.1931,Z 191,A 22.1781,B 0.9928,C 0.0243,E1 1.1439,E2 432.0597} C_DIS
LIN {X 130.0598,Y 44.8735,Z 191,A 20.2967,B 0.9928,C 0.0281,E1 1.1456,E2 433.8832} C_DIS
LIN {X 131.178,Y 41.4923,Z 191,A 18.9949,B 0.9926,C 0.0312,E1 1.1467,E2 435.1631} C_DIS
LIN {X 132.0841,Y 38.5092,Z 191,A 17.8663,B 0.9926,C 0.0339,E1 1.1476,E2 436.2712} C_DIS
LIN {X 132.9957,Y 35.2328,Z 191,A 16.6235,B 0.9924,C 0.0368,E1 1.1485,E2 437.493} C_DIS
LIN {X 133.8062,Y 32.0173,Z 191,A 15.3967,B 0.9924,C 0.0398,E1 1.1493,E2 438.7012} C_DIS
LIN {X 134.6323,Y 28.3513,Z 191,A 14.0446,B 0.9922,C 0.043,E1 1.1501,E2 440.0274} C_DIS
LIN {X 135.3181,Y 24.8718,Z 191,A 12.2949,B 0.9919,C 0.0485,E1 1.151,E2 441.8118} C_DIS
LIN {X 136.0408,Y 20.5514,Z 191,A 11.2082,B 0.9919,C 0.0497,E1 1.1515,E2 442.8067} C_DIS
LIN {X 136.5706,Y 16.6678,Z 191,A 9.3411,B 0.9916,C 0.0554,E1 1.1521,E2 444.7043} C_DIS
LIN {X 136.9914,Y 12.7568,Z 191,A 8.2247,B 0.9915,C 0.0572,E1 1.1524,E2 445.7554} C_DIS
LIN {X 137.4528,Y 6.0368,Z 191,A 5.8564,B 0.9911,C 0.0628,E1 1.1528,E2 448.0694} C_DIS
LIN {X 137.5564,Y 2.7845,Z 191,A 4.2134,B 0.9908,C 0.0681,E1 1.1529,E2 449.75} C_DIS
LIN {X 137.5775,Y -1.4988,Z 191,A 3.0781,B 0.9907,C 0.0696,E1 1.1529,E2 450.8031} C_DIS
LIN {X 137.4312,Y -6.4873,Z 191,A 1.3571,B 0.9904,C 0.0735,E1 1.1528,E2 452.479} C_DIS
LIN {X 137.218,Y -10.0226,Z 191,A -0.092,B 0.9901,C 0.0774,E1 1.1525,E2 453.9256} C_DIS
LIN {X 136.9084,Y -13.6213,Z 191,A -1.339,B 0.9899,C 0.0803,E1 1.1522,E2 455.1401} C_DIS
LIN {X 136.5553,Y -16.7959,Z 191,A -2.9154,B 0.9894,C 0.0853,E1 1.1516,E2 456.7494} C_DIS
LIN {X 136.0169,Y -20.7054,Z 191,A -3.8611,B 0.9894,C 0.0861,E1 1.1513,E2 457.6048} C_DIS
LIN {X 135.4711,Y -24.0172,Z 191,A -5.2542,B 0.989,C 0.0899,E1 1.1507,E2 458.9982} C_DIS
LIN {X 134.7817,Y -27.6244,Z 191,A -6.6092,B 0.9887,C 0.0932,E1 1.1499,E2 460.3312} C_DIS
LIN {X 134.0208,Y -31.11,Z 191,A -7.8746,B 0.9885,C 0.0961,E1 1.1492,E2 461.5684} C_DIS
LIN {X 133.0231,Y -35.13,Z 191,A -9.4164,B 0.9881,C 0.0998,E1 1.1481,E2 463.0871} C_DIS
LIN {X 132.0785,Y -38.5283,Z 191,A -10.7105,B 0.9878,C 0.1029,E1 1.1471,E2 464.3588} C_DIS
LIN {X 130.8702,Y -42.4555,Z 191,A -12.4475,B 0.9873,C 0.1076,E1 1.1457,E2 466.1005} C_DIS
LIN {X 129.8042,Y -45.6107,Z 191,A -13.3938,B 0.9871,C 0.109,E1 1.1449,E2 466.9889} C_DIS
LIN {X 128.6922,Y -48.6581,Z 191,A -14.6459,B 0.9868,C 0.112,E1 1.1436,E2 468.2286} C_DIS
LIN {X 127.4906,Y -51.7238,Z 191,A -15.7881,B 0.9865,C 0.1145,E1 1.1425,E2 469.3409} C_DIS
LIN {X 125.9612,Y -55.3494,Z 191,A -17.2542,B 0.9861,C 0.1178,E1 1.1409,E2 470.785} C_DIS
LIN {X 124.7852,Y -57.9466,Z 191,A -18.3351,B 0.9858,C 0.1204,E1 1.1397,E2 471.8522} C_DIS
LIN {X 123.2711,Y -61.1015,Z 191,A -19.6247,B 0.9854,C 0.1232,E1 1.1381,E2 473.1201} C_DIS
LIN {X 121.21,Y -65.0983,Z 191,A -21.2581,B 0.985,C 0.1268,E1 1.136,E2 474.7224} C_DIS
LIN {X 119.4697,Y -68.2396,Z 191,A -22.684,B 0.9845,C 0.1302,E1 1.1341,E2 476.1398} C_DIS
LIN {X 115.9202,Y -74.1092,Z 191,A -25.0096,B 0.984,C 0.1345,E1 1.1308,E2 478.3948} C_DIS
LIN {X 112.6852,Y -78.9421,Z 191,A -27.1433,B 0.9833,C 0.139,E1 1.1275,E2 480.4906} C_DIS
LIN {X 109.7148,Y -83.0197,Z 191,A -29.2852,B 0.9826,C 0.1442,E1 1.1239,E2 482.6399} C_DIS
LIN {X 107.781,Y -85.5157,Z 191,A -30.4292,B 0.9823,C 0.1464,E1 1.122,E2 483.7614} C_DIS
LIN {X 104.9742,Y -88.9389,Z 191,A -32.0755,B 0.9818,C 0.1496,E1 1.1191,E2 485.3817} C_DIS
LIN {X 102.0554,Y -92.2735,Z 191,A -33.7657,B 0.9813,C 0.153,E1 1.116,E2 487.0516} C_DIS
LIN {X 99.3068,Y -95.2253,Z 191,A -35.205,B 0.9809,C 0.1555,E1 1.1132,E2 488.4587} C_DIS
LIN {X 96.4659,Y -98.102,Z 191,A -36.7712,B 0.9804,C 0.1586,E1 1.1102,E2 490.0099} C_DIS
LIN {X 93.1889,Y -101.22,Z 191,A -38.4567,B 0.9799,C 0.1616,E1 1.1068,E2 491.669} C_DIS
LIN {X 89.8255,Y -104.2162,Z 191,A -40.1205,B 0.9794,C 0.1645,E1 1.1033,E2 493.3044} C_DIS
LIN {X 86.6777,Y -106.8493,Z 191,A -41.7439,B 0.9789,C 0.1675,E1 1.0998,E2 494.9171} C_DIS
LIN {X 83.0663,Y -109.68,Z 191,A -43.4597,B 0.9784,C 0.1703,E1 1.096,E2 496.6069} C_DIS
LIN {X 79.4951,Y -112.2953,Z 191,A -45.1416,B 0.9779,C 0.1731,E1 1.0923,E2 498.2674} C_DIS
LIN {X 75.1502,Y -115.2483,Z 191,A -47.1469,B 0.9774,C 0.1763,E1 1.0876,E2 500.2485} C_DIS
LIN {X 71.4673,Y -117.5677,Z 191,A -48.8168,B 0.9769,C 0.1788,E1 1.0837,E2 501.8994} C_DIS
LIN {X 65.3898,Y -121.0534,Z 191,A -51.4917,B 0.9762,C 0.1826,E1 1.0772,E2 504.5419} C_DIS
LIN {X 62.1429,Y -122.7495,Z 191,A -52.8419,B 0.9759,C 0.1843,E1 1.0739,E2 505.8682} C_DIS
LIN {X 58.2361,Y -124.6513,Z 191,A -54.5731,B 0.9754,C 0.1868,E1 1.0695,E2 507.5895} C_DIS
LIN {X 55.2082,Y -126.0222,Z 191,A -56.4911,B 0.9746,C 0.191,E1 1.0643,E2 509.5847} C_DIS
LIN {X 49.7893,Y -128.2581,Z 191,A -57.7493,B 0.9748,C 0.1896,E1 1.0615,E2 510.6753} C_DIS
LIN {X 46.3155,Y -129.5536,Z 191,A -59.5365,B 0.9743,C 0.1926,E1 1.0567,E2 512.4987} C_DIS
LIN {X 43.1039,Y -130.6573,Z 191,A -60.8361,B 0.974,C 0.194,E1 1.0532,E2 513.7828} C_DIS
LIN {X 39.9528,Y -131.6549,Z 191,A -62.1657,B 0.9737,C 0.1954,E1 1.0496,E2 515.1066} C_DIS
LIN {X 35.6899,Y -132.8738,Z 191,A -63.9056,B 0.9734,C 0.1972,E1 1.045,E2 516.8323} C_DIS
LIN {X 32.2056,Y -133.7608,Z 191,A -65.3305,B 0.9731,C 0.1985,E1 1.0411,E2 518.2478} C_DIS
LIN {X 28.2646,Y -134.6506,Z 191,A -67.2222,B 0.9726,C 0.2009,E1 1.0358,E2 520.1708} C_DIS
LIN {X 24.7812,Y -135.3343,Z 191,A -68.203,B 0.9726,C 0.2005,E1 1.0332,E2 521.0807} C_DIS
LIN {X 16.9552,Y -136.5363,Z 191,A -71.7891,B 0.9719,C 0.2042,E1 1.0231,E2 524.7106} C_DIS
LIN {X 13.5239,Y -136.9177,Z 191,A -73.1333,B 0.9717,C 0.2049,E1 1.0193,E2 526.0422} C_DIS
LIN {X 10.2692,Y -137.2,Z 191,A -73.9617,B 0.9719,C 0.2041,E1 1.0172,E2 526.7942} C_DIS
LIN {X 6.1176,Y -137.4494,Z 191,A -75.9691,B 0.9715,C 0.206,E1 1.0114,E2 528.8427} C_DIS
LIN {X 0.9755,Y -137.5796,Z 191,A -77.8854,B 0.9715,C 0.2064,E1 1.0061,E2 530.7273} C_DIS
Enddeposition()
LIN {X 0.9755,Y -137.5796,Z 191,A -77.8854,B 0.9715,C 0.2064,E1 1.0061,E2 530.7273} C_DIS
Startdeposition()
$VEL.CP = VEL_PRINT
LIN {X 3.0738,Y -138.4506,Z 191,A -76.4374,B 0.9637,C 0.2043,E1 1.0022,E2 529.2207} C_DIS
LIN {X 6.3371,Y -138.3388,Z 191,A -75.015,B 0.9639,C 0.2033,E1 1.0063,E2 527.787} C_DIS
LIN {X 10.0899,Y -138.1144,Z 191,A -73.6781,B 0.9639,C 0.203,E1 1.01,E2 526.4814} C_DIS
LIN {X 12.9298,Y -137.8778,Z 191,A -72.4709,B 0.9641,C 0.2021,E1 1.0134,E2 525.2693} C_DIS
LIN {X 16.098,Y -137.5439,Z 191,A -71.1993,B 0.9643,C 0.2013,E1 1.0169,E2 524.0038} C_DIS
LIN {X 19.2832,Y -137.1336,Z 191,A -70.0926,B 0.9643,C 0.201,E1 1.0199,E2 522.9289} C_DIS
LIN {X 22.4828,Y -136.6454,Z 191,A -68.6365,B 0.9647,C 0.1995,E1 1.0241,E2 521.4548} C_DIS
LIN {X 25.1991,Y -136.1728,Z 191,A -67.5461,B 0.9649,C 0.1986,E1 1.0271,E2 520.3711} C_DIS
LIN {X 28.4184,Y -135.5375,Z 191,A -66.2511,B 0.9651,C 0.1975,E1 1.0306,E2 519.0845} C_DIS
LIN {X 32.1413,Y -134.701,Z 191,A -64.749,B 0.9654,C 0.1961,E1 1.0347,E2 517.5926} C_DIS
LIN {X 34.8744,Y -134.0216,Z 191,A -63.5096,B 0.9657,C 0.1946,E1 1.0382,E2 516.3416} C_DIS
LIN {X 38.4152,Y -133.0483,Z 191,A -62.1533,B 0.9659,C 0.1935,E1 1.0418,E2 515.0081} C_DIS
LIN {X 41.8301,Y -132.0138,Z 191,A -60.9916,B 0.966,C 0.1929,E1 1.0448,E2 513.8914} C_DIS
LIN {X 44.5573,Y -131.1208,Z 191,A -59.5646,B 0.9665,C 0.1905,E1 1.0487,E2 512.4286} C_DIS
LIN {X 48.2656,Y -129.7992,Z 191,A -58.2346,B 0.9667,C 0.1895,E1 1.0521,E2 511.1411} C_DIS
LIN {X 50.9755,Y -128.7615,Z 191,A -57.0492,B 0.967,C 0.1879,E1 1.0552,E2 509.9571} C_DIS
LIN {X 54.1638,Y -127.4531,Z 191,A -55.7133,B 0.9673,C 0.1862,E1 1.0587,E2 508.6333} C_DIS
LIN {X 57.7524,Y -125.8654,Z 191,A -54.3615,B 0.9676,C 0.185,E1 1.0621,E2 507.3199} C_DIS
LIN {X 60.482,Y -124.579,Z 191,A -53.0498,B 0.968,C 0.1828,E1 1.0654,E2 505.998} C_DIS
LIN {X 63.7113,Y -122.9581,Z 191,A -51.6441,B 0.9684,C 0.1808,E1 1.0689,E2 504.6042} C_DIS
LIN {X 67.469,Y -120.9378,Z 191,A -49.9248,B 0.9689,C 0.1781,E1 1.0732,E2 502.8903} C_DIS
LIN {X 71.2816,Y -118.7306,Z 191,A -48.2468,B 0.9693,C 0.1756,E1 1.0772,E2 501.232} C_DIS
LIN {X 75.126,Y -116.3358,Z 191,A -46.6053,B 0.9697,C 0.1733,E1 1.081,E2 499.6227} C_DIS
LIN {X 78.5021,Y -114.0844,Z 191,A -45.0722,B 0.9702,C 0.1708,E1 1.0845,E2 498.1093} C_DIS
LIN {X 81.851,Y -111.7061,Z 191,A -43.5525,B 0.9706,C 0.1685,E1 1.0879,E2 496.6143} C_DIS
LIN {X 84.8764,Y -109.4249,Z 191,A -42.0756,B 0.971,C 0.1658,E1 1.0912,E2 495.1492} C_DIS
LIN {X 88.2829,Y -106.6955,Z 191,A -40.4184,B 0.9715,C 0.1629,E1 1.0948,E2 493.5119} C_DIS
LIN {X 91.594,Y -103.8672,Z 191,A -38.7977,B 0.972,C 0.1601,E1 1.0982,E2 491.9158} C_DIS
LIN {X 94.7042,Y -101.0402,Z 191,A -37.224,B 0.9724,C 0.1572,E1 1.1014,E2 490.3644} C_DIS
LIN {X 97.7278,Y -98.1179,Z 191,A -35.6672,B 0.9729,C 0.1544,E1 1.1044,E2 488.8324} C_DIS
LIN {X 100.851,Y -94.9048,Z 191,A -34.0144,B 0.9734,C 0.1513,E1 1.1076,E2 487.2067} C_DIS
LIN {X 103.4566,Y -92.0584,Z 191,A -32.5546,B 0.9738,C 0.1484,E1 1.1103,E2 485.7652} C_DIS
LIN {X 106.1582,Y -88.9284,Z 191,A -31.0392,B 0.9743,C 0.1455,E1 1.113,E2 484.276} C_DIS
LIN {X 108.8003,Y -85.6758,Z 191,A -29.4741,B 0.9748,C 0.1423,E1 1.1157,E2 482.7335} C_DIS
LIN {X 111.3409,Y -82.3481,Z 191,A -27.9827,B 0.9752,C 0.1394,E1 1.1182,E2 481.2746} C_DIS
LIN {X 113.5781,Y -79.2329,Z 191,A -26.5145,B 0.9756,C 0.1362,E1 1.1205,E2 479.8219} C_DIS
LIN {X 116.0054,Y -75.6349,Z 191,A -24.8985,B 0.9761,C 0.1327,E1 1.123,E2 478.2298} C_DIS
LIN {X 118.2735,Y -72.0374,Z 191,A -23.3529,B 0.9765,C 0.1295,E1 1.1252,E2 476.7127} C_DIS
LIN {X 120.5068,Y -68.2358,Z 191,A -21.6842,B 0.977,C 0.1257,E1 1.1275,E2 475.0643} C_DIS
LIN {X 122.3682,Y -64.8346,Z 191,A -20.3312,B 0.9774,C 0.123,E1 1.1293,E2 473.7451} C_DIS
LIN {X 124.0446,Y -61.5654,Z 191,A -19.0272,B 0.9777,C 0.1202,E1 1.1309,E2 472.4698} C_DIS
LIN {X 125.3297,Y -58.9108,Z 191,A -17.9489,B 0.978,C 0.1178,E1 1.1321,E2 471.4103} C_DIS
LIN {X 126.7668,Y -55.7512,Z 191,A -16.6817,B 0.9784,C 0.1149,E1 1.1335,E2 470.1653} C_DIS
LIN {X 128.118,Y -52.5717,Z 191,A -15.3125,B 0.9788,C 0.1115,E1 1.135,E2 468.8034} C_DIS
LIN {X 129.5798,Y -48.8513,Z 191,A -14.1044,B 0.979,C 0.1095,E1 1.1362,E2 467.6551} C_DIS
LIN {X 130.7347,Y -45.671,Z 191,A -12.7334,B 0.9794,C 0.1059,E1 1.1375,E2 466.2871} C_DIS
LIN {X 131.6572,Y -42.9464,Z 191,A -11.5616,B 0.9797,C 0.1028,E1 1.1385,E2 465.1171} C_DIS
LIN {X 132.8117,Y -39.2231,Z 191,A -10.2701,B 0.98,C 0.1002,E1 1.1395,E2 463.8681} C_DIS
LIN {X 133.742,Y -35.9228,Z 191,A -9.2087,B 0.9802,C 0.0982,E1 1.1402,E2 462.8541} C_DIS
LIN {X 134.4316,Y -33.2591,Z 191,A -7.903,B 0.9806,C 0.0942,E1 1.1412,E2 461.5251} C_DIS
LIN {X 135.2965,Y -29.5346,Z 191,A -6.6384,B 0.9808,C 0.0916,E1 1.1419,E2 460.3023} C_DIS
LIN {X 135.9599,Y -26.3127,Z 191,A -5.4157,B 0.9811,C 0.0886,E1 1.1426,E2 459.0972} C_DIS
LIN {X 136.477,Y -23.4924,Z 191,A -4.3125,B 0.9813,C 0.0858,E1 1.1431,E2 458.0045} C_DIS
LIN {X 136.9756,Y -20.3888,Z 191,A -3.2671,B 0.9815,C 0.0835,E1 1.1435,E2 456.9925} C_DIS
LIN {X 137.4126,Y -17.1983,Z 191,A -2.1008,B 0.9818,C 0.0807,E1 1.1439,E2 455.8475} C_DIS
LIN {X 137.7728,Y -14.0239,Z 191,A -0.8478,B 0.982,C 0.0774,E1 1.1443,E2 454.6028} C_DIS
LIN {X 138.0792,Y -10.5717,Z 191,A 0.3836,B 0.9823,C 0.0745,E1 1.1446,E2 453.3974} C_DIS
LIN {X 138.2928,Y -7.253,Z 191,A 1.513,B 0.9824,C 0.072,E1 1.1447,E2 452.2998} C_DIS
LIN {X 138.4208,Y -4.1446,Z 191,A 2.6386,B 0.9826,C 0.0693,E1 1.1449,E2 451.1948} C_DIS
LIN {X 138.4824,Y -0.6319,Z 191,A 3.8681,B 0.9828,C 0.0665,E1 1.1449,E2 449.9939} C_DIS
LIN {X 138.4585,Y 2.5998,Z 191,A 5.1324,B 0.9831,C 0.0631,E1 1.1449,E2 448.7384} C_DIS
LIN {X 138.326,Y 6.5928,Z 191,A 6.5484,B 0.9833,C 0.0598,E1 1.1447,E2 447.3525} C_DIS
LIN {X 138.137,Y 9.7808,Z 191,A 7.6947,B 0.9834,C 0.057,E1 1.1445,E2 446.2283} C_DIS
LIN {X 137.8778,Y 12.9298,Z 191,A 8.8422,B 0.9836,C 0.0542,E1 1.1442,E2 445.1009} C_DIS
LIN {X 137.5439,Y 16.098,Z 191,A 9.9992,B 0.9837,C 0.0514,E1 1.1439,E2 443.964} C_DIS
LIN {X 136.9756,Y 20.3888,Z 191,A 11.6922,B 0.984,C 0.047,E1 1.1432,E2 442.2828} C_DIS
LIN {X 136.3718,Y 24.0871,Z 191,A 12.7739,B 0.984,C 0.0452,E1 1.1427,E2 441.2605} C_DIS
LIN {X 135.8652,Y 26.8077,Z 191,A 13.9391,B 0.9842,C 0.0419,E1 1.1421,E2 440.0922} C_DIS
LIN {X 135.1894,Y 30.0308,Z 191,A 15.2602,B 0.9843,C 0.0384,E1 1.1413,E2 438.7759} C_DIS
LIN {X 134.2793,Y 33.8591,Z 191,A 16.5697,B 0.9844,C 0.0356,E1 1.1405,E2 437.5062} C_DIS
LIN {X 133.1391,Y 38.1052,Z 191,A 18.168,B 0.9846,C 0.0318,E1 1.1393,E2 435.9352} C_DIS
LIN {X 132.0138,Y 41.8301,Z 191,A 19.5727,B 0.9846,C 0.0285,E1 1.1382,E2 434.5557} C_DIS
LIN {X 130.9706,Y 44.9903,Z 191,A 20.8125,B 0.9847,C 0.0255,E1 1.1371,E2 433.3326} C_DIS
LIN {X 129.7992,Y 48.2656,Z 191,A 21.898,B 0.9847,C 0.0235,E1 1.1361,E2 432.2908} C_DIS
LIN {X 128.6034,Y 51.3676,Z 191,A 23.2735,B 0.9849,C 0.0198,E1 1.1347,E2 430.915} C_DIS
LIN {X 127.2419,Y 54.6523,Z 191,A 24.4074,B 0.9849,C 0.0176,E1 1.1335,E2 429.8225} C_DIS
LIN {X 125.958,Y 57.552,Z 191,A 25.6595,B 0.9849,C 0.0145,E1 1.1321,E2 428.5774} C_DIS
LIN {X 124.579,Y 60.482,Z 191,A 26.921,B 0.985,C 0.0114,E1 1.1306,E2 427.3253} C_DIS
LIN {X 122.8413,Y 63.9338,Z 191,A 28.3325,B 0.985,C 0.0082,E1 1.1288,E2 425.9363} C_DIS
LIN {X 120.9378,Y 67.469,Z 191,A 29.9164,B 0.985,C 0.0044,E1 1.1267,E2 424.3616} C_DIS
LIN {X 118.6466,Y 71.4204,Z 191,A 31.557,B 0.985,C 0.0009,E1 1.1244,E2 422.7511} C_DIS
LIN {X 116.3938,Y 75.0367,Z 191,A 33.1065,B 0.985,C -0.0025,E1 1.1221,E2 421.2272} C_DIS
LIN {X 114.0844,Y 78.5021,Z 191,A 34.6129,B 0.985,C -0.0056,E1 1.1198,E2 419.7468} C_DIS
LIN {X 111.6049,Y 81.9888,Z 191,A 36.2169,B 0.985,C -0.0091,E1 1.1172,E2 418.1625} C_DIS
LIN {X 109.1822,Y 85.1896,Z 191,A 37.6991,B 0.985,C -0.0122,E1 1.1147,E2 416.7016} C_DIS
LIN {X 106.5524,Y 88.4558,Z 191,A 39.257,B 0.985,C -0.0154,E1 1.112,E2 415.1646} C_DIS
LIN {X 103.8672,Y 91.594,Z 191,A 40.7778,B 0.985,C -0.0184,E1 1.1092,E2 413.6661} C_DIS
LIN {X 101.0402,Y 94.7042,Z 191,A 42.3839,B 0.9848,C -0.0217,E1 1.1062,E2 412.0756} C_DIS
LIN {X 97.863,Y 97.9835,Z 191,A 44.0747,B 0.9848,C -0.0249,E1 1.1029,E2 410.4083} C_DIS
LIN {X 94.7042,Y 101.0402,Z 191,A 45.6769,B 0.9847,C -0.0279,E1 1.0997,E2 408.8315} C_DIS
LIN {X 91.594,Y 103.8672,Z 191,A 47.2566,B 0.9846,C -0.0308,E1 1.0964,E2 407.2705} C_DIS
LIN {X 88.4558,Y 106.5524,Z 191,A 48.7909,B 0.9846,C -0.0336,E1 1.0931,E2 405.7566} C_DIS
LIN {X 85.1896,Y 109.1822,Z 191,A 50.3074,B 0.9844,C -0.0361,E1 1.0899,E2 404.2656} C_DIS
LIN {X 82.1643,Y 111.4759,Z 191,A 51.8011,B 0.9844,C -0.0388,E1 1.0865,E2 402.7809} C_DIS
LIN {X 78.7276,Y 113.9297,Z 191,A 53.385,B 0.9842,C -0.0414,E1 1.0829,E2 401.216} C_DIS
LIN {X 75.5227,Y 116.0782,Z 191,A 54.8691,B 0.9842,C -0.0439,E1 1.0795,E2 399.745} C_DIS
LIN {X 71.5142,Y 118.5899,Z 191,A 56.609,B 0.984,C -0.0465,E1 1.0753,E2 398.0301} C_DIS
LIN {X 67.9998,Y 120.6394,Z 191,A 58.2139,B 0.9839,C -0.049,E1 1.0714,E2 396.4344} C_DIS
LIN {X 64.0826,Y 122.7631,Z 191,A 59.8134,B 0.9838,C -0.0511,E1 1.0675,E2 394.8629} C_DIS
LIN {X 61.5654,Y 124.0446,Z 191,A 60.8997,B 0.9837,C -0.0527,E1 1.0648,E2 393.7862} C_DIS
LIN {X 58.5819,Y 125.4818,Z 191,A 62.21,B 0.9836,C -0.0545,E1 1.0615,E2 392.4829} C_DIS
LIN {X 55.7512,Y 126.7668,Z 191,A 63.4931,B 0.9835,C -0.0564,E1 1.0582,E2 391.2004} C_DIS
LIN {X 52.0601,Y 128.3243,Z 191,A 64.911,B 0.9834,C -0.058,E1 1.0546,E2 389.8099} C_DIS
LIN {X 49.3755,Y 129.3834,Z 191,A 66.0157,B 0.9833,C -0.0593,E1 1.0517,E2 388.7155} C_DIS
LIN {X 45.671,Y 130.7347,Z 191,A 67.5405,B 0.9832,C -0.0611,E1 1.0477,E2 387.203} C_DIS
LIN {X 42.3688,Y 131.8417,Z 191,A 68.8714,B 0.9831,C -0.0625,E1 1.0441,E2 385.8847} C_DIS
LIN {X 39.2231,Y 132.8117,Z 191,A 70.1717,B 0.9831,C -0.0639,E1 1.0406,E2 384.5917} C_DIS
LIN {X 35.9928,Y 133.7234,Z 191,A 71.4742,B 0.9829,C -0.0653,E1 1.0371,E2 383.2992} C_DIS
LIN {X 32.7738,Y 134.5486,Z 191,A 72.7912,B 0.9829,C -0.0666,E1 1.0335,E2 381.989} C_DIS
LIN {X 29.5346,Y 135.2965,Z 191,A 74.0846,B 0.9827,C -0.0677,E1 1.03,E2 380.7051} C_DIS
LIN {X 26.3127,Y 135.9599,Z 191,A 75.3658,B 0.9827,C -0.0688,E1 1.0265,E2 379.4331} C_DIS
LIN {X 23.5928,Y 136.4602,Z 191,A 76.6043,B 0.9826,C -0.0701,E1 1.023,E2 378.1845} C_DIS
LIN {X 20.3888,Y 136.9756,Z 191,A 77.881,B 0.9826,C -0.071,E1 1.0195,E2 376.9156} C_DIS
LIN {X 17.1983,Y 137.4126,Z 191,A 79.0304,B 0.9825,C -0.0716,E1 1.0163,E2 375.7869} C_DIS
LIN {X 14.0239,Y 137.7728,Z 191,A 80.301,B 0.9825,C -0.0724,E1 1.0127,E2 374.5225} C_DIS
LIN {X 10.8679,Y 138.0576,Z 191,A 81.5653,B 0.9824,C -0.0732,E1 1.0092,E2 373.2637} C_DIS
LIN {X 7.253,Y 138.2928,Z 191,A 83.0597,B 0.9823,C -0.0741,E1 1.005,E2 371.7703} C_DIS
LIN {X 4.0942,Y 138.4222,Z 191,A 84.3217,B 0.9823,C -0.0746,E1 1.0014,E2 370.5138} C_DIS
LIN {X 0,Y 138.4847,Z 191,A 85.9359,B 0.9823,C -0.0752,E1 0.9969,E2 368.9091} C_DIS
LIN {X -3.2871,Y 138.4447,Z 191,A 87.1928,B 0.9822,C -0.0756,E1 0.9934,E2 367.664} C_DIS
LIN {X -6.1737,Y 138.347,Z 191,A 88.5828,B 0.9822,C -0.0764,E1 0.9894,E2 366.2531} C_DIS
LIN {X -9.9779,Y 138.1226,Z 191,A 90.0343,B 0.9822,C -0.0765,E1 0.9853,E2 364.8159} C_DIS
LIN {X -12.9548,Y 137.8754,Z 191,A 91.2247,B 0.9821,C -0.0767,E1 0.982,E2 363.631} C_DIS
LIN {X -16.098,Y 137.5439,Z 191,A 92.5315,B 0.9821,C -0.0769,E1 0.9783,E2 362.3248} C_DIS
LIN {X -19.2832,Y 137.1336,Z 191,A 93.6723,B 0.9821,C -0.0766,E1 0.9752,E2 361.2053} C_DIS
LIN {X -22.4828,Y 136.6454,Z 191,A 95.1987,B 0.9821,C -0.077,E1 0.9708,E2 359.6589} C_DIS
LIN {X -25.1991,Y 136.1728,Z 191,A 96.4531,B 0.9821,C -0.0771,E1 0.9673,E2 358.3927} C_DIS
LIN {X -28.4184,Y 135.5375,Z 191,A 97.7117,B 0.9821,C -0.0768,E1 0.9638,E2 357.1456} C_DIS
LIN {X -32.1413,Y 134.701,Z 191,A 99.3094,B 0.9821,C -0.0765,E1 0.9594,E2 355.5465} C_DIS
LIN {X -34.8744,Y 134.0216,Z 191,A 100.4921,B 0.9821,C -0.0763,E1 0.9562,E2 354.3625} C_DIS
LIN {X -38.1052,Y 133.1391,Z 191,A 101.9879,B 0.9821,C -0.076,E1 0.9521,E2 352.8553} C_DIS
LIN {X -41.8301,Y 132.0138,Z 191,A 103.35,B 0.9822,C -0.075,E1 0.9485,E2 351.5211} C_DIS
LIN {X -44.5573,Y 131.1208,Z 191,A 104.9225,B 0.9822,C -0.075,E1 0.9441,E2 349.907} C_DIS
LIN {X -48.2656,Y 129.7992,Z 191,A 106.389,B 0.9823,C -0.0739,E1 0.9403,E2 348.459} C_DIS
LIN {X -51.4604,Y 128.566,Z 191,A 107.7095,B 0.9823,C -0.0729,E1 0.9368,E2 347.1499} C_DIS
LIN {X -54.1638,Y 127.4531,Z 191,A 109.168,B 0.9824,C -0.0724,E1 0.933,E2 345.6647} C_DIS
LIN {X -57.3337,Y 126.0589,Z 191,A 110.7992,B 0.9824,C -0.0715,E1 0.9287,E2 344.0124} C_DIS
LIN {X -60.482,Y 124.579,Z 191,A 112.1663,B 0.9826,C -0.0703,E1 0.9252,E2 342.6541} C_DIS
LIN {X -63.6053,Y 123.0137,Z 191,A 113.8209,B 0.9826,C -0.0692,E1 0.921,E2 340.9771} C_DIS
LIN {X -67.469,Y 120.9378,Z 191,A 115.7318,B 0.9828,C -0.0675,E1 0.9163,E2 339.0566} C_DIS
LIN {X -71.2816,Y 118.7306,Z 191,A 117.5992,B 0.9828,C -0.0656,E1 0.9117,E2 337.1851} C_DIS
LIN {X -74.9669,Y 116.4384,Z 191,A 119.5224,B 0.983,C -0.0636,E1 0.9071,E2 335.2488} C_DIS
LIN {X -78.5021,Y 114.0844,Z 191,A 121.3594,B 0.9832,C -0.0615,E1 0.9028,E2 333.4039} C_DIS
LIN {X -81.851,Y 111.7061,Z 191,A 123.1473,B 0.9832,C -0.0593,E1 0.8987,E2 331.607} C_DIS
LIN {X -84.7012,Y 109.5608,Z 191,A 124.8097,B 0.9834,C -0.0574,E1 0.8949,E2 329.9245} C_DIS
LIN {X -88.0551,Y 106.8842,Z 191,A 126.7782,B 0.9836,C -0.0548,E1 0.8905,E2 327.9353} C_DIS
LIN {X -91.3875,Y 104.0497,Z 191,A 128.6347,B 0.9837,C -0.052,E1 0.8866,E2 326.0746} C_DIS
LIN {X -94.2503,Y 101.4629,Z 191,A 130.451,B 0.9838,C -0.0495,E1 0.8828,E2 324.2343} C_DIS
LIN {X -97.3441,Y 98.4991,Z 191,A 132.4475,B 0.984,C -0.0465,E1 0.8787,E2 322.2134} C_DIS
LIN {X -100.4253,Y 95.356,Z 191,A 134.3347,B 0.9841,C -0.0433,E1 0.875,E2 320.3198} C_DIS
LIN {X -102.8591,Y 92.7255,Z 191,A 135.9763,B 0.9842,C -0.0406,E1 0.8718,E2 318.6608} C_DIS
LIN {X -105.4007,Y 89.825,Z 191,A 137.7492,B 0.9844,C -0.0375,E1 0.8685,E2 316.8685} C_DIS
LIN {X -107.9015,Y 86.8051,Z 191,A 139.5986,B 0.9844,C -0.0343,E1 0.8652,E2 314.9938} C_DIS
LIN {X -110.2712,Y 83.7752,Z 191,A 141.3395,B 0.9846,C -0.031,E1 0.8622,E2 313.2366} C_DIS
LIN {X -112.3912,Y 80.9088,Z 191,A 143.0711,B 0.9846,C -0.0279,E1 0.8593,E2 311.476} C_DIS
LIN {X -114.7772,Y 77.4857,Z 191,A 144.9817,B 0.9848,C -0.0241,E1 0.8562,E2 309.5448} C_DIS
LIN {X -117.1173,Y 73.901,Z 191,A 147.0153,B 0.9848,C -0.0201,E1 0.8531,E2 307.4814} C_DIS
LIN {X -119.3199,Y 70.2895,Z 191,A 149.0451,B 0.9849,C -0.016,E1 0.8501,E2 305.4196} C_DIS
LIN {X -121.6546,Y 66.1664,Z 191,A 151.0017,B 0.985,C -0.0114,E1 0.8474,E2 303.4647} C_DIS
LIN {X -123.0137,Y 63.6053,Z 191,A 152.6822,B 0.985,C -0.0083,E1 0.8452,E2 301.7276} C_DIS
LIN {X -124.81,Y 59.9985,Z 191,A 154.2099,B 0.985,C -0.0044,E1 0.8433,E2 300.2176} C_DIS
LIN {X -126.0589,Y 57.3337,Z 191,A 155.8372,B 0.985,C -0.0011,E1 0.8414,E2 298.542} C_DIS
LIN {X -127.4531,Y 54.1638,Z 191,A 157.4842,B 0.985,C 0.0026,E1 0.8395,E2 296.8699} C_DIS
LIN {X -128.9021,Y 50.6138,Z 191,A 159.3322,B 0.985,C 0.0068,E1 0.8375,E2 294.9911} C_DIS
LIN {X -130.0972,Y 47.458,Z 191,A 160.9836,B 0.985,C 0.0106,E1 0.8359,E2 293.3094} C_DIS
LIN {X -131.2859,Y 44.0616,Z 191,A 162.4195,B 0.985,C 0.0144,E1 0.8346,E2 291.8809} C_DIS
LIN {X -132.3243,Y 40.8372,Z 191,A 164.283,B 0.985,C 0.0184,E1 0.833,E2 289.9615} C_DIS
LIN {X -133.2871,Y 37.5759,Z 191,A 165.8926,B 0.9848,C 0.0223,E1 0.8317,E2 288.3277} C_DIS
LIN {X -134.0216,Y 34.8744,Z 191,A 167.2491,B 0.9848,C 0.0256,E1 0.8307,E2 286.9475} C_DIS
LIN {X -134.9342,Y 31.1479,Z 191,A 169.0952,B 0.9846,C 0.0301,E1 0.8295,E2 285.0699} C_DIS
LIN {X -135.6383,Y 27.9228,Z 191,A 170.6859,B 0.9845,C 0.034,E1 0.8286,E2 283.4519} C_DIS
LIN {X -136.2163,Y 24.956,Z 191,A 172.1275,B 0.9844,C 0.0376,E1 0.8278,E2 281.9871} C_DIS
LIN {X -136.804,Y 21.4968,Z 191,A 173.6216,B 0.9842,C 0.0416,E1 0.8271,E2 280.4885} C_DIS
LIN {X -137.2038,Y 18.7917,Z 191,A 175.1603,B 0.984,C 0.0451,E1 0.8265,E2 278.8989} C_DIS
LIN {X -137.6022,Y 15.609,Z 191,A 176.7108,B 0.9839,C 0.049,E1 0.826,E2 277.3208} C_DIS
LIN {X -137.9522,Y 12.1162,Z 191,A 178.4787,B 0.9836,C 0.0534,E1 0.8255,E2 275.5134} C_DIS
LIN {X -138.1722,Y 9.2976,Z 191,A 179.9372,B 0.9834,C 0.0569,E1 0.8252,E2 274.0184} C_DIS
LIN {X -138.3657,Y 5.6958,Z 191,A -178.4786,B 0.9832,C 0.0611,E1 0.825,E2 272.4232} C_DIS
LIN {X -138.4585,Y 2.5998,Z 191,A -176.9144,B 0.9829,C 0.065,E1 0.825,E2 270.8231} C_DIS
LIN {X -138.4824,Y -0.6319,Z 191,A -175.2764,B 0.9827,C 0.069,E1 0.825,E2 269.1467} C_DIS
LIN {X -138.3915,Y -5.0337,Z 191,A -173.454,B 0.9823,C 0.0741,E1 0.825,E2 267.3252} C_DIS
LIN {X -138.239,Y -8.2143,Z 191,A -171.7255,B 0.982,C 0.0781,E1 0.8253,E2 265.5436} C_DIS
LIN {X -138.0166,Y -11.3528,Z 191,A -170.1988,B 0.9817,C 0.0819,E1 0.8256,E2 263.9879} C_DIS
LIN {X -137.7203,Y -14.5117,Z 191,A -168.6391,B 0.9813,C 0.0858,E1 0.8261,E2 262.3961} C_DIS
LIN {X -137.3238,Y -17.8761,Z 191,A -167.0373,B 0.981,C 0.0898,E1 0.8266,E2 260.7685} C_DIS
LIN {X -136.9509,Y -20.5485,Z 191,A -165.6012,B 0.9807,C 0.0931,E1 0.8272,E2 259.2904} C_DIS
LIN {X -136.3718,Y -24.0871,Z 191,A -164.1946,B 0.9803,C 0.0971,E1 0.8279,E2 257.8947} C_DIS
LIN {X -135.8652,Y -26.8077,Z 191,A -162.493,B 0.9799,C 0.1007,E1 0.8288,E2 256.1191} C_DIS
LIN {X -135.0676,Y -30.5638,Z 191,A -160.7584,B 0.9795,C 0.1051,E1 0.8299,E2 254.3655} C_DIS
LIN {X -134.0216,Y -34.8744,Z 191,A -158.6474,B 0.9789,C 0.1102,E1 0.8313,E2 252.2181} C_DIS
LIN {X -132.9856,Y -38.6292,Z 191,A -156.7884,B 0.9784,C 0.1146,E1 0.8328,E2 250.326} C_DIS
LIN {X -132.0138,Y -41.8301,Z 191,A -155.1506,B 0.9779,C 0.1183,E1 0.8342,E2 248.6542} C_DIS
LIN {X -131.1208,Y -44.5573,Z 191,A -153.6216,B 0.9775,C 0.1216,E1 0.8356,E2 247.0789} C_DIS
LIN {X -129.7992,Y -48.2656,Z 191,A -152.1367,B 0.977,C 0.1257,E1 0.837,E2 245.6143} C_DIS
LIN {X -128.7615,Y -50.9755,Z 191,A -150.5268,B 0.9766,C 0.1289,E1 0.8387,E2 243.9486} C_DIS
LIN {X -127.4531,Y -54.1638,Z 191,A -148.8858,B 0.9761,C 0.1325,E1 0.8405,E2 242.2783} C_DIS
LIN {X -126.0589,Y -57.3337,Z 191,A -147.2408,B 0.9756,C 0.1361,E1 0.8424,E2 240.6044} C_DIS
LIN {X -124.3887,Y -60.8678,Z 191,A -145.3495,B 0.9751,C 0.1401,E1 0.8447,E2 238.6754} C_DIS
LIN {X -122.7631,Y -64.0826,Z 191,A -143.6821,B 0.9745,C 0.1437,E1 0.8469,E2 236.9837} C_DIS
LIN {X -120.6394,Y -67.9998,Z 191,A -141.549,B 0.9739,C 0.148,E1 0.8498,E2 234.8106} C_DIS
LIN {X -118.4799,Y -71.6961,Z 191,A -139.5155,B 0.9733,C 0.152,E1 0.8528,E2 232.7407} C_DIS
LIN {X -116.3938,Y -75.0367,Z 191,A -137.665,B 0.9727,C 0.1555,E1 0.8556,E2 230.8594} C_DIS
LIN {X -114.0844,Y -78.5021,Z 191,A -135.7256,B 0.9721,C 0.1592,E1 0.8587,E2 228.8897} C_DIS
LIN {X -111.7061,Y -81.851,Z 191,A -133.8924,B 0.9716,C 0.1627,E1 0.8618,E2 227.0377} C_DIS
LIN {X -109.5608,Y -84.7012,Z 191,A -132.1723,B 0.9711,C 0.1656,E1 0.8648,E2 225.2831} C_DIS
LIN {X -106.9421,Y -87.9852,Z 191,A -130.2,B 0.9705,C 0.1689,E1 0.8683,E2 223.2776} C_DIS
LIN {X -104.0497,Y -91.3875,Z 191,A -128.2592,B 0.9699,C 0.1724,E1 0.8719,E2 221.3237} C_DIS
LIN {X -101.2835,Y -94.443,Z 191,A -126.3227,B 0.9694,C 0.1753,E1 0.8757,E2 219.3541} C_DIS
LIN {X -98.5552,Y -97.2877,Z 191,A -124.5839,B 0.9688,C 0.1781,E1 0.8791,E2 217.5999} C_DIS
LIN {X -95.8045,Y -99.9967,Z 191,A -122.7661,B 0.9684,C 0.1806,E1 0.8828,E2 215.7504} C_DIS
LIN {X -92.7255,Y -102.8591,Z 191,A -120.8103,B 0.9679,C 0.1832,E1 0.887,E2 213.7633} C_DIS
LIN {X -89.353,Y -105.8019,Z 191,A -118.8584,B 0.9674,C 0.1859,E1 0.8912,E2 211.7969} C_DIS
LIN {X -86.1394,Y -108.4335,Z 191,A -117.0042,B 0.9669,C 0.1882,E1 0.8953,E2 209.9229} C_DIS
LIN {X -82.5682,Y -111.1771,Z 191,A -115.0182,B 0.9665,C 0.1906,E1 0.8998,E2 207.919} C_DIS
LIN {X -79.2329,Y -113.5781,Z 191,A -113.1844,B 0.9661,C 0.1926,E1 0.9041,E2 206.0656} C_DIS
LIN {X -75.7642,Y -115.9214,Z 191,A -111.2793,B 0.9657,C 0.1945,E1 0.9086,E2 204.135} C_DIS
LIN {X -72.0374,Y -118.2735,Z 191,A -109.4061,B 0.9653,C 0.1964,E1 0.9131,E2 202.2543} C_DIS
LIN {X -68.2358,Y -120.5068,Z 191,A -107.4205,B 0.965,C 0.198,E1 0.9181,E2 200.2448} C_DIS
LIN {X -65.1564,Y -122.1992,Z 191,A -106.0235,B 0.9647,C 0.1994,E1 0.9215,E2 198.8558} C_DIS
LIN {X -61.6728,Y -123.9916,Z 191,A -104.2969,B 0.9644,C 0.2006,E1 0.9259,E2 197.1133} C_DIS
LIN {X -58.9108,Y -125.3297,Z 191,A -102.8557,B 0.9643,C 0.2014,E1 0.9297,E2 195.6467} C_DIS
LIN {X -55.5655,Y -126.8471,Z 191,A -101.3378,B 0.9641,C 0.2024,E1 0.9336,E2 194.1288} C_DIS
LIN {X -52.0805,Y -128.316,Z 191,A -99.8131,B 0.9638,C 0.2035,E1 0.9375,E2 192.6094} C_DIS
LIN {X -49.3755,Y -129.3834,Z 191,A -98.5739,B 0.9637,C 0.2041,E1 0.9408,E2 191.3647} C_DIS
LIN {X -45.671,Y -130.7347,Z 191,A -96.9012,B 0.9635,C 0.2049,E1 0.9453,E2 189.6854} C_DIS
LIN {X -42.9464,Y -131.6572,Z 191,A -95.5381,B 0.9635,C 0.205,E1 0.949,E2 188.2964} C_DIS
LIN {X -39.2231,Y -132.8117,Z 191,A -94.0438,B 0.9633,C 0.2058,E1 0.953,E2 186.819} C_DIS
LIN {X -35.9455,Y -133.736,Z 191,A -92.6085,B 0.9633,C 0.2062,E1 0.957,E2 185.3793} C_DIS
LIN {X -33.2591,Y -134.4316,Z 191,A -91.3127,B 0.9633,C 0.2062,E1 0.9606,E2 184.0614} C_DIS
LIN {X -29.5346,Y -135.2965,Z 191,A -89.8624,B 0.9632,C 0.2067,E1 0.9645,E2 182.6299} C_DIS
LIN {X -26.3127,Y -135.9599,Z 191,A -88.6789,B 0.963,C 0.2072,E1 0.9677,E2 181.472} C_DIS
LIN {X -23.5928,Y -136.4602,Z 191,A -87.216,B 0.9632,C 0.2065,E1 0.972,E2 179.9616} C_DIS
LIN {X -20.0131,Y -137.0293,Z 191,A -85.9949,B 0.9631,C 0.2071,E1 0.9753,E2 178.7809} C_DIS
LIN {X -17.1983,Y -137.4126,Z 191,A -84.6915,B 0.9631,C 0.2067,E1 0.979,E2 177.4582} C_DIS
LIN {X -14.0239,Y -137.7728,Z 191,A -83.3832,B 0.9631,C 0.2065,E1 0.9826,E2 176.1512} C_DIS
LIN {X -10.2678,Y -138.1014,Z 191,A -81.8954,B 0.9632,C 0.2063,E1 0.9868,E2 174.6733} C_DIS
LIN {X -7.0595,Y -138.3025,Z 191,A -80.582,B 0.9633,C 0.206,E1 0.9905,E2 173.3617} C_DIS
LIN {X -4.1446,Y -138.4208,Z 191,A -79.3548,B 0.9634,C 0.2055,E1 0.994,E2 172.1309} C_DIS
LIN {X -1.0616,Y -138.4788,Z 191,A -78.0622,B 0.9635,C 0.2049,E1 0.9977,E2 170.8351} C_DIS
LIN {X -1.0616,Y -138.4788,Z 191,A -78.0622,B 0.9635,C 0.2049,E1 0.9977,E2 170.8351} C_DIS
Enddeposition()
LIN {X 0.9891,Y -139.3743,Z 191,A -77.339,B 0.9559,C 0.2049,E1 0.992,E2 170.1561} C_DIS
Startdeposition()
$VEL.CP = VEL_PRINT
LIN {X -1.7905,Y -139.371,Z 191,A -78.9513,B 0.9555,C 0.2069,E1 0.9872,E2 171.8388} C_DIS
LIN {X -5.6058,Y -139.2688,Z 191,A -80.4396,B 0.9554,C 0.2072,E1 0.9831,E2 173.3159} C_DIS
LIN {X -9.6684,Y -139.0465,Z 191,A -82.0963,B 0.9553,C 0.2076,E1 0.9784,E2 174.9711} C_DIS
LIN {X -12.8269,Y -138.7908,Z 191,A -83.4113,B 0.9553,C 0.208,E1 0.9747,E2 176.2886} C_DIS
LIN {X -16.5982,Y -138.3895,Z 191,A -84.8217,B 0.9553,C 0.2078,E1 0.9708,E2 177.6777} C_DIS
LIN {X -19.6162,Y -137.9941,Z 191,A -86.1171,B 0.9553,C 0.208,E1 0.9671,E2 178.9803} C_DIS
LIN {X -22.8521,Y -137.4952,Z 191,A -87.503,B 0.9552,C 0.2082,E1 0.9632,E2 180.3726} C_DIS
LIN {X -26.7505,Y -136.7914,Z 191,A -89.2581,B 0.9552,C 0.2084,E1 0.9583,E2 182.1471} C_DIS
LIN {X -31.0644,Y -135.8753,Z 191,A -91.3172,B 0.9551,C 0.2087,E1 0.9525,E2 184.2432} C_DIS
LIN {X -34.7343,Y -134.9846,Z 191,A -92.5966,B 0.9553,C 0.2077,E1 0.9491,E2 185.483} C_DIS
LIN {X -38.9736,Y -133.8215,Z 191,A -94.2902,B 0.9554,C 0.2069,E1 0.9445,E2 187.1605} C_DIS
LIN {X -45.0451,Y -131.9031,Z 191,A -97.1282,B 0.9556,C 0.2063,E1 0.9368,E2 190.032} C_DIS
LIN {X -48.8824,Y -130.528,Z 191,A -98.6117,B 0.9558,C 0.2051,E1 0.9329,E2 191.4876} C_DIS
LIN {X -51.2722,Y -129.6106,Z 191,A -100.0311,B 0.9558,C 0.2051,E1 0.929,E2 192.9615} C_DIS
LIN {X -55.0491,Y -128.0497,Z 191,A -101.5774,B 0.9561,C 0.2038,E1 0.9251,E2 194.4884} C_DIS
LIN {X -58.248,Y -126.6266,Z 191,A -103.0339,B 0.9563,C 0.2028,E1 0.9213,E2 195.9478} C_DIS
LIN {X -61.3782,Y -125.1393,Z 191,A -104.5685,B 0.9565,C 0.2019,E1 0.9173,E2 197.4989} C_DIS
LIN {X -66.3024,Y -122.604,Z 191,A -107.0057,B 0.9569,C 0.2001,E1 0.9112,E2 199.9602} C_DIS
LIN {X -69.8688,Y -120.6066,Z 191,A -108.7983,B 0.9572,C 0.1986,E1 0.9067,E2 201.7695} C_DIS
LIN {X -73.7467,Y -118.2753,Z 191,A -110.7867,B 0.9576,C 0.1967,E1 0.9019,E2 203.7769} C_DIS
LIN {X -77.5892,Y -115.7911,Z 191,A -112.7327,B 0.958,C 0.1946,E1 0.8973,E2 205.7326} C_DIS
LIN {X -80.8626,Y -113.5293,Z 191,A -114.5346,B 0.9584,C 0.1928,E1 0.8931,E2 207.5589} C_DIS
LIN {X -84.4532,Y -110.8843,Z 191,A -116.5201,B 0.9589,C 0.1905,E1 0.8885,E2 209.5667} C_DIS
LIN {X -87.8193,Y -108.2383,Z 191,A -118.4439,B 0.9593,C 0.1882,E1 0.8842,E2 211.5142} C_DIS
LIN {X -91.5678,Y -105.0854,Z 191,A -120.5986,B 0.9599,C 0.1853,E1 0.8796,E2 213.6893} C_DIS
LIN {X -94.7611,Y -102.2156,Z 191,A -122.4333,B 0.9604,C 0.1825,E1 0.8757,E2 215.5341} C_DIS
LIN {X -99.8632,Y -97.2373,Z 191,A -125.7799,B 0.9613,C 0.1778,E1 0.8689,E2 218.9406} C_DIS
LIN {X -103.0143,Y -93.8922,Z 191,A -127.8663,B 0.9619,C 0.1745,E1 0.8649,E2 221.0552} C_DIS
LIN {X -105.6424,Y -90.9246,Z 191,A -129.6159,B 0.9624,C 0.1715,E1 0.8616,E2 222.8217} C_DIS
LIN {X -108.5651,Y -87.4141,Z 191,A -131.7171,B 0.9631,C 0.168,E1 0.8578,E2 224.9545} C_DIS
LIN {X -110.5341,Y -84.9112,Z 191,A -133.6277,B 0.9635,C 0.1655,E1 0.8544,E2 226.9503} C_DIS
LIN {X -113.1636,Y -81.374,Z 191,A -135.2553,B 0.9641,C 0.1617,E1 0.8517,E2 228.5515} C_DIS
LIN {X -115.7259,Y -77.6868,Z 191,A -137.3375,B 0.9648,C 0.1578,E1 0.8484,E2 230.6667} C_DIS
LIN {X -118.0387,Y -74.1253,Z 191,A -139.0969,B 0.9654,C 0.154,E1 0.8457,E2 232.4277} C_DIS
LIN {X -119.9638,Y -70.9681,Z 191,A -141.0369,B 0.9659,C 0.1506,E1 0.8428,E2 234.4264} C_DIS
LIN {X -122.2106,Y -67.0244,Z 191,A -143.0998,B 0.9666,C 0.1462,E1 0.84,E2 236.5164} C_DIS
LIN {X -124.0292,Y -63.5921,Z 191,A -144.8571,B 0.9672,C 0.1425,E1 0.8377,E2 238.2955} C_DIS
LIN {X -125.6593,Y -60.3061,Z 191,A -146.5648,B 0.9677,C 0.1388,E1 0.8355,E2 240.0305} C_DIS
LIN {X -126.9736,Y -57.4904,Z 191,A -148.1531,B 0.9681,C 0.1356,E1 0.8336,E2 241.6616} C_DIS
LIN {X -128.3598,Y -54.3251,Z 191,A -149.8006,B 0.9686,C 0.132,E1 0.8318,E2 243.34} C_DIS
LIN {X -129.7913,Y -50.8074,Z 191,A -151.4493,B 0.9692,C 0.128,E1 0.8301,E2 245.0001} C_DIS
LIN {X -132.4853,Y -43.3049,Z 191,A -155.3496,B 0.9703,C 0.1193,E1 0.8264,E2 248.9846} C_DIS
LIN {X -133.6148,Y -39.6795,Z 191,A -157.1373,B 0.9708,C 0.115,E1 0.8249,E2 250.8026} C_DIS
LIN {X -134.664,Y -35.954,Z 191,A -158.8174,B 0.9713,C 0.1107,E1 0.8236,E2 252.494} C_DIS
LIN {X -135.4554,Y -32.8475,Z 191,A -160.3693,B 0.9717,C 0.1071,E1 0.8226,E2 254.077} C_DIS
LIN {X -136.2068,Y -29.5779,Z 191,A -161.8897,B 0.9721,C 0.1033,E1 0.8216,E2 255.6158} C_DIS
LIN {X -136.8548,Y -26.4188,Z 191,A -163.5348,B 0.9725,C 0.0994,E1 0.8207,E2 257.3032} C_DIS
LIN {X -137.3797,Y -23.544,Z 191,A -165.3454,B 0.9729,C 0.0956,E1 0.8198,E2 259.1946} C_DIS
LIN {X -137.9008,Y -20.269,Z 191,A -166.6781,B 0.9733,C 0.0919,E1 0.8192,E2 260.5225} C_DIS
LIN {X -138.3711,Y -16.7529,Z 191,A -168.3331,B 0.9736,C 0.0877,E1 0.8186,E2 262.2028} C_DIS
LIN {X -138.7511,Y -13.2396,Z 191,A -169.9447,B 0.974,C 0.0836,E1 0.8182,E2 263.8346} C_DIS
LIN {X -139.0875,Y -9.0599,Z 191,A -172.6318,B 0.9745,C 0.0779,E1 0.8177,E2 266.647} C_DIS
LIN {X -139.3101,Y -4.5033,Z 191,A -174.3187,B 0.9749,C 0.0728,E1 0.8175,E2 268.3084} C_DIS
LIN {X -139.3377,Y 3.5094,Z 191,A -177.8726,B 0.9755,C 0.0634,E1 0.8175,E2 271.8943} C_DIS
LIN {X -138.974,Y 10.6608,Z 191,A 178.3047,B 0.9761,C 0.0544,E1 0.8181,E2 275.8284} C_DIS
LIN {X -138.6907,Y 13.8689,Z 191,A 175.8497,B 0.9763,C 0.0496,E1 0.8189,E2 278.4254} C_DIS
LIN {X -137.8796,Y 20.4169,Z 191,A 173.4115,B 0.9767,C 0.0424,E1 0.8198,E2 280.8277} C_DIS
LIN {X -136.9968,Y 25.6759,Z 191,A 171.0807,B 0.9769,C 0.0362,E1 0.8209,E2 283.1745} C_DIS
LIN {X -136.3773,Y 28.7882,Z 191,A 169.6955,B 0.977,C 0.0326,E1 0.8217,E2 284.569} C_DIS
LIN {X -135.3541,Y 33.2681,Z 191,A 166.9366,B 0.9772,C 0.0267,E1 0.8236,E2 287.4344} C_DIS
LIN {X -134.3554,Y 37.0936,Z 191,A 165.5033,B 0.9773,C 0.0226,E1 0.8246,E2 288.8431} C_DIS
LIN {X -133.3945,Y 40.4121,Z 191,A 163.8085,B 0.9774,C 0.0186,E1 0.826,E2 290.5707} C_DIS
LIN {X -132.2919,Y 43.8856,Z 191,A 162.0527,B 0.9774,C 0.0145,E1 0.8275,E2 292.357} C_DIS
LIN {X -130.3519,Y 49.3526,Z 191,A 159.7501,B 0.9776,C 0.0084,E1 0.8297,E2 294.6482} C_DIS
LIN {X -126.8629,Y 57.737,Z 191,A 154.987,B 0.9776,C -0.0017,E1 0.835,E2 299.5338} C_DIS
LIN {X -126.8629,Y 57.737,Z 191,A 154.9859,B 0.9776,C -0.0017,E1 0.835,E2 299.535} C_DIS
LIN {X -125.2046,Y 61.2459,Z 191,A 153.3003,B 0.9776,C -0.0056,E1 0.837,E2 301.2303} C_DIS
LIN {X -123.5619,Y 64.4949,Z 191,A 151.4758,B 0.9776,C -0.0094,E1 0.8394,E2 303.0929} C_DIS
LIN {X -121.4851,Y 68.3299,Z 191,A 149.4788,B 0.9775,C -0.0137,E1 0.8422,E2 305.1129} C_DIS
LIN {X -118.9459,Y 72.6605,Z 191,A 147.0057,B 0.9775,C -0.0186,E1 0.8458,E2 307.6327} C_DIS
LIN {X -116.5037,Y 76.5148,Z 191,A 144.8977,B 0.9773,C -0.0228,E1 0.849,E2 309.7666} C_DIS
LIN {X -113.9911,Y 80.2101,Z 191,A 141.9116,B 0.9773,C -0.0271,E1 0.8541,E2 312.8836} C_DIS
LIN {X -110.0378,Y 85.553,Z 191,A 139.7707,B 0.9771,C -0.0325,E1 0.8576,E2 314.9553} C_DIS
LIN {X -107.2842,Y 88.9815,Z 191,A 137.7489,B 0.9769,C -0.0361,E1 0.8612,E2 317.0006} C_DIS
LIN {X -104.275,Y 92.4898,Z 191,A 135.6196,B 0.9768,C -0.0398,E1 0.8652,E2 319.1548} C_DIS
LIN {X -101.3274,Y 95.7097,Z 191,A 133.6747,B 0.9766,C -0.043,E1 0.869,E2 321.1157} C_DIS
LIN {X -98.2056,Y 98.9104,Z 191,A 131.6869,B 0.9766,C -0.0462,E1 0.8729,E2 323.1193} C_DIS
LIN {X -95.2682,Y 101.7433,Z 191,A 129.751,B 0.9764,C -0.049,E1 0.877,E2 325.0832} C_DIS
LIN {X -92.0909,Y 104.6277,Z 191,A 127.8274,B 0.9762,C -0.0517,E1 0.881,E2 327.0237} C_DIS
LIN {X -88.5763,Y 107.6197,Z 191,A 125.7624,B 0.9761,C -0.0545,E1 0.8855,E2 329.1063} C_DIS
LIN {X -85.0367,Y 110.438,Z 191,A 123.7546,B 0.9759,C -0.0571,E1 0.89,E2 331.1293} C_DIS
LIN {X -82.0907,Y 112.6448,Z 191,A 121.5305,B 0.9759,C -0.0588,E1 0.8953,E2 333.431} C_DIS
LIN {X -77.686,Y 115.7264,Z 191,A 119.8642,B 0.9756,C -0.0618,E1 0.899,E2 335.0363} C_DIS
LIN {X -71.0027,Y 119.9431,Z 191,A 116.0858,B 0.9754,C -0.0651,E1 0.9082,E2 338.8712} C_DIS
LIN {X -67.9581,Y 121.694,Z 191,A 114.7722,B 0.9754,C -0.0666,E1 0.9114,E2 340.1697} C_DIS
LIN {X -63.8372,Y 123.9044,Z 191,A 112.9295,B 0.9752,C -0.0685,E1 0.916,E2 342.0025} C_DIS
LIN {X -61.3553,Y 125.1506,Z 191,A 111.5524,B 0.9752,C -0.0692,E1 0.9196,E2 343.4048} C_DIS
LIN {X -57.2491,Y 127.0815,Z 191,A 109.9387,B 0.975,C -0.0709,E1 0.9236,E2 344.9899} C_DIS
LIN {X -52.3664,Y 129.17,Z 191,A 107.4688,B 0.975,C -0.0721,E1 0.9302,E2 347.4901} C_DIS
LIN {X -49.1161,Y 130.4405,Z 191,A 106.0512,B 0.9749,C -0.0729,E1 0.9339,E2 348.9051} C_DIS
LIN {X -46.2403,Y 131.4887,Z 191,A 104.7037,B 0.9749,C -0.0735,E1 0.9375,E2 350.2618} C_DIS
LIN {X -42.6582,Y 132.693,Z 191,A 103.1661,B 0.9748,C -0.0742,E1 0.9416,E2 351.7968} C_DIS
LIN {X -39.5641,Y 133.6486,Z 191,A 101.796,B 0.9748,C -0.0746,E1 0.9454,E2 353.1705} C_DIS
LIN {X -36.7291,Y 134.4573,Z 191,A 100.3747,B 0.9748,C -0.0746,E1 0.9493,E2 354.614} C_DIS
LIN {X -32.8795,Y 135.4477,Z 191,A 99.0051,B 0.9747,C -0.0755,E1 0.953,E2 355.954} C_DIS
LIN {X -26.4515,Y 136.8485,Z 191,A 95.3715,B 0.9747,C -0.0742,E1 0.9633,E2 359.6866} C_DIS
LIN {X -20.5313,Y 137.8631,Z 191,A 93.6071,B 0.9747,C -0.0755,E1 0.968,E2 361.3743} C_DIS
LIN {X -14.1345,Y 138.665,Z 191,A 90.9026,B 0.9747,C -0.075,E1 0.9757,E2 364.0835} C_DIS
LIN {X -10.0498,Y 139.0186,Z 191,A 89.3926,B 0.9747,C -0.075,E1 0.9799,E2 365.5737} C_DIS
LIN {X -6.2561,Y 139.2429,Z 191,A 87.6787,B 0.9747,C -0.0742,E1 0.9847,E2 367.3035} C_DIS
LIN {X -2.0552,Y 139.3666,Z 191,A 86.0655,B 0.9748,C -0.0738,E1 0.9893,E2 368.9036} C_DIS
LIN {X 2.1648,Y 139.3648,Z 191,A 84.4368,B 0.9748,C -0.0732,E1 0.9938,E2 370.5201} C_DIS
LIN {X 5.8151,Y 139.2606,Z 191,A 82.9242,B 0.9749,C -0.0724,E1 0.9981,E2 372.0334} C_DIS
LIN {X 9.6136,Y 139.0505,Z 191,A 81.4115,B 0.9749,C -0.0715,E1 1.0024,E2 373.54} C_DIS
LIN {X 13.3648,Y 138.7391,Z 191,A 80.0798,B 0.975,C -0.071,E1 1.0061,E2 374.8475} C_DIS
LIN {X 15.9006,Y 138.4727,Z 191,A 78.9165,B 0.975,C -0.07,E1 1.0094,E2 376.0232} C_DIS
LIN {X 19.4311,Y 138.0205,Z 191,A 77.6196,B 0.9751,C -0.0692,E1 1.0129,E2 377.3014} C_DIS
LIN {X 22.4635,Y 137.56,Z 191,A 76.1247,B 0.9753,C -0.0675,E1 1.0172,E2 378.8216} C_DIS
LIN {X 26.4842,Y 136.8423,Z 191,A 74.2283,B 0.9754,C -0.0652,E1 1.0225,E2 380.7413} C_DIS
LIN {X 31.1857,Y 135.8476,Z 191,A 72.8934,B 0.9754,C -0.0652,E1 1.026,E2 382.0054} C_DIS
LIN {X 34.8072,Y 134.9661,Z 191,A 71.3509,B 0.9755,C -0.0635,E1 1.0302,E2 383.5487} C_DIS
LIN {X 37.6176,Y 134.2088,Z 191,A 69.8925,B 0.9757,C -0.0612,E1 1.0343,E2 385.0357} C_DIS
LIN {X 41.7305,Y 132.9893,Z 191,A 68.5699,B 0.9757,C -0.0605,E1 1.0377,E2 386.3093} C_DIS
LIN {X 45.3015,Y 131.8142,Z 191,A 67.1941,B 0.9758,C -0.0591,E1 1.0413,E2 387.6658} C_DIS
LIN {X 48.4906,Y 130.6748,Z 191,A 65.8301,B 0.9759,C -0.0574,E1 1.0449,E2 389.0265} C_DIS
LIN {X 51.9615,Y 129.3332,Z 191,A 64.5103,B 0.9759,C -0.056,E1 1.0484,E2 390.3225} C_DIS
LIN {X 55.0458,Y 128.0511,Z 191,A 63.1814,B 0.9761,C -0.0541,E1 1.0518,E2 391.6462} C_DIS
LIN {X 58.8852,Y 126.3319,Z 191,A 61.7616,B 0.9761,C -0.0526,E1 1.0554,E2 393.0309} C_DIS
LIN {X 63.0823,Y 124.2887,Z 191,A 59.911,B 0.9763,C -0.0499,E1 1.06,E2 394.8735} C_DIS
LIN {X 66.3187,Y 122.5952,Z 191,A 58.3229,B 0.9765,C -0.0471,E1 1.064,E2 396.4714} C_DIS
LIN {X 70.3601,Y 120.3209,Z 191,A 56.6166,B 0.9765,C -0.0446,E1 1.0681,E2 398.1548} C_DIS
LIN {X 74.0724,Y 118.0721,Z 191,A 54.9997,B 0.9767,C -0.0421,E1 1.0719,E2 399.7525} C_DIS
LIN {X 77.6799,Y 115.7305,Z 191,A 53.3448,B 0.9768,C -0.0393,E1 1.0758,E2 401.3945} C_DIS
LIN {X 81.7428,Y 112.8969,Z 191,A 51.5121,B 0.9769,C -0.0363,E1 1.0799,E2 403.2037} C_DIS
LIN {X 85.322,Y 110.2168,Z 191,A 49.8583,B 0.977,C -0.0335,E1 1.0836,E2 404.8362} C_DIS
LIN {X 88.3943,Y 107.7688,Z 191,A 48.3156,B 0.9771,C -0.0305,E1 1.0869,E2 406.3707} C_DIS
LIN {X 92.076,Y 104.6409,Z 191,A 45.7079,B 0.9773,C -0.0237,E1 1.0926,E2 409.0499} C_DIS
LIN {X 97.608,Y 99.5001,Z 191,A 43.79,B 0.9773,C -0.0223,E1 1.0962,E2 410.8309} C_DIS
Enddeposition()
END
